// TIA Portal V16 program export: 11 tag tables, 23 data types, 17 data blocks, 38 code blocks (in call order from the OBs), 10 instance data blocks

VAR_GLOBAL   // PLC tag table "CONST"
END_VAR
VAR_GLOBAL CONSTANT   // user constants
   MAX_STEP_NUMB : Int := 50;
   MIN_STEP_NUMB : Int := 1;
   MAX_DEV_NUMB : Int := 16;
   MIN_DEV_NUMB : Int := 1;
   UF_CM_STANDBY : Int := 0;
   UF_CM_FILTRATION : Int := 2;
   UF_CM_START : Int := 1;
   UF_CM_HW : Int := 4;
   UF_CM_HW_A : Int := 5;
   UF_CM_CEB1 : Int := 6;
   UF_CM_CEB1_A : Int := 7;
   UF_CM_CEB2 : Int := 8;
   UF_CM_CEB2_A : Int := 9;
   UF_CM_STOP : Int := 3;
END_VAR

VAR_GLOBAL   // PLC tag table "Default tag table"
   System_Byte AT %MB1 : Byte;
   FirstScan AT %M1.0 : Bool;
   DiagStatusUpdate AT %M1.1 : Bool;
   AlwaysTRUE AT %M1.2 : Bool;
   AlwaysFALSE AT %M1.3 : Bool;
   Clock_Byte AT %MB0 : Byte;
   Clock_10Hz AT %M0.0 : Bool;
   Clock_5Hz AT %M0.1 : Bool;
   "Clock_2.5Hz" AT %M0.2 : Bool;
   Clock_2Hz AT %M0.3 : Bool;
   "Clock_1.25Hz" AT %M0.4 : Bool;
   Clock_1Hz AT %M0.5 : Bool;
   "Clock_0.625Hz" AT %M0.6 : Bool;
   "Clock_0.5Hz" AT %M0.7 : Bool;
   ClockOneSycle AT %MB2 : Byte;
   ClockOneCycle10HZ AT %M2.0 : Bool;
   ClockOneCycle5HZ AT %M2.1 : Bool;
   ClockOneCycle2_5HZ AT %M2.2 : Bool;
   ClockOneCycle2HZ AT %M2.3 : Bool;
   ClockOneCycle1_25HZ AT %M2.4 : Bool;
   ClockOneCycle1HZ AT %M2.5 : Bool;
   ClockOneCycle0_65HZ AT %M2.6 : Bool;
   ClockOneCycle0_5HZ AT %M2.7 : Bool;
END_VAR

VAR_GLOBAL   // PLC tag table "HW"
   PLC_RAW_DI AT %I0.0 : "PLC_HW_DI";
   PLC_RAW_DQ AT %Q0.0 : "PLC_HW_DQ";
   PLC_RAW_AI AT %I64.0 : "PLC_HW_AI";
   PLC_RAW_AQ AT %Q64.0 : "PLC_HW_AQ";
   ET_RAW_DI AT %I2.0 : "ET_HW_DI";
   ET_RAW_DQ AT %Q2.0 : "ET_HW_DQ";
   ET_RAW_AI AT %I68.0 : "ET_HW_AI";
   ET_RAW_AQ AT %Q68.0 : "ET_HW_AQ";
END_VAR
VAR_GLOBAL CONSTANT   // user constants
   PLC_DI : Int := 13;
   PLC_DQ : Int := 9;
   PLC_AI : Int := 1;
   PLC_AQ : Int := 1;
   ET_DI : Int := 79;
   ET_DQ : Int := 31;
   ET_AI : Int := 39;
   ET_AQ : Int := 7;
END_VAR

VAR_GLOBAL   // PLC tag table "A1_AI"
   aiDVA503_Pos AT %IW64 : Int;   // DVA503 Завдання
   aiDVA510_Pos AT %IW66 : Int;   // DVA510 Завдання
END_VAR
VAR_GLOBAL CONSTANT   // user constants
   "iwDVA-503_Setting" : Int := 0;
   "iwDVA-510_Setting" : Int := 1;
END_VAR

VAR_GLOBAL   // PLC tag table "A1_AQ"
   AO_DVA503_Setting AT %QW64 : Int;   // DVA503 Стан
   AO_DVA510_Setting AT %QW66 : Int;   // DVA510 Стан
END_VAR
VAR_GLOBAL CONSTANT   // user constants
   "qwDVA-503_Setting" : Int := 0;
   "qw_DVA-510_Setting" : Int := 1;
END_VAR

VAR_GLOBAL   // PLC tag table "A1_DI"
   iP301_Run AT %I0.0 : Bool;   // P301 Робота
   iP302_Run AT %I0.1 : Bool;   // P302 Робота
   iP1201_Run AT %I0.2 : Bool;   // P1201 Робота
   iP1202_Run AT %I0.3 : Bool;   // P1202 Робота
   iP1501_Run AT %I0.4 : Bool;   // P1501 Робота
   iP1502_Run AT %I0.5 : Bool;   // P1502 Робота
   iP70x_Ready AT %I0.6 : Bool;   // P70x Готовність
   iP701_Run AT %I0.7 : Bool;   // P701 Робота
   iP702_Run AT %I1.0 : Bool;   // P702 Робота
   iP201_Ready AT %I1.1 : Bool;   // P201 Готовність
   iP201_Run AT %I1.2 : Bool;   // P201 Робота
   iC501_Ready AT %I1.3 : Bool;   // C501 Готовність
   iStop AT %I1.4 : Bool;   // Аварійне вимикання
   iSF_Fail AT %I1.5 : Bool;   // Аварія захисних автоматів
END_VAR
VAR_GLOBAL CONSTANT   // user constants
   "iP-301_Run" : Int := 0;
   "iP-302_Run" : Int := 1;
   "iP-1201_Run" : Int := 2;
   "iP-1202_Run" : Int := 3;
   "iP-1501_Run" : Int := 4;
   "iP-1502_Run" : Int := 5;
   "iP-70x_Ready" : Int := 6;
   "iP-701_Run" : Int := 7;
   "iP-702_Run" : Int := 8;
   "iP-201_Ready" : Int := 9;
   "iP-201_Run" : Int := 10;
   "iC-501_Ready" : Int := 11;
   i_Stop : Int := 12;
   i_SF_Fail : Int := 13;
END_VAR

VAR_GLOBAL   // PLC tag table "A1_DQ"
   Tag_1 AT %Q0.0 : Bool;
   qP301_Start AT %Q0.1 : Bool;   // P301 Пуск
   qP302_Start AT %Q0.2 : Bool;   // P302 Пуск
   qP1201_Start AT %Q0.3 : Bool;   // P1201 Пуск
   qP1202_Start AT %Q0.4 : Bool;   // P1202 Пуск
   qP1501_Start AT %Q0.5 : Bool;   // P1501 Пуск
   qP1502_Start AT %Q0.6 : Bool;   // P1502 Пуск
   qP701_Start AT %Q0.7 : Bool;   // P701 Пуск
   qP702_Start AT %Q1.0 : Bool;   // P702 Пуск
   qP2001_Start AT %Q1.1 : Bool;   // P2001 Пуск
END_VAR
VAR_GLOBAL CONSTANT   // user constants
   iTag_1 : Int := 0;
   "qP-301_Start" : Int := 1;
   "qP-302_Start" : Int := 2;
   "qP-1201_Start" : Int := 3;
   "qP-1202_Start" : Int := 4;
   "qP-1501_Start" : Int := 5;
   "qP-1502_Start" : Int := 6;
   "qP-701_Start" : Int := 7;
   "qP-702_Start" : Int := 8;
   "qP-2001_Start" : Int := 9;
END_VAR

VAR_GLOBAL   // PLC tag table "A10_AI"
   aiLT201 AT %IW68 : Int;   // Рівень ємності TW201 LT201
   aiLT202 AT %IW70 : Int;   // Рівень ємності TW202 LT202
   aiPT301 AT %IW72 : Int;   // Тиск PS3 PT301
   aiPT401 AT %IW74 : Int;   // Тиск MDF4 PT401
   aiPT501 AT %IW76 : Int;   // Тиск повітря UF PT501
   aiPT502 AT %IW78 : Int;   // Тиск вхідної води UF PT502
   aiPT503 AT %IW80 : Int;   // Тиск фільтрата UF PT503
   aiPT504 AT %IW82 : Int;   // Тиск стічних вод UF PT504
   aiPT505 AT %IW84 : Int;   // Тиск вхідної води UF PT505
   aiPT506 AT %IW86 : Int;   // Тиск фільтрата UF PT506
   aiPT507 AT %IW88 : Int;   // Тиск стічних вод UF PT507
   aiLT601 AT %IW90 : Int;   // Рівень ємності TW601 LT601
   aiPT701 AT %IW92 : Int;   // Тиск PS7 PT701
   aiPT901 AT %IW94 : Int;   // Тиск насоса RO PT901
   aiPT902 AT %IW96 : Int;   // Тиск концентрата RO PT902
   aiLT1101 AT %IW98 : Int;   // Рівень ємності TW1101 LT1101
   aiPT1201 AT %IW100 : Int;   // Тиск PS12 PT1201
   aiPT1301 AT %IW102 : Int;   // Тиск насоса NF PT1301
   aiPT1302 AT %IW104 : Int;   // Тиск концентрата NF PT1302
   aiLT1401 AT %IW106 : Int;   // Рівень ємності TW1401 LT1401
   aiLT1402 AT %IW108 : Int;   // Рівень ємності TW1402 LT1402
   aiPT1501 AT %IW110 : Int;   // Тиск PS15 PT1501
   aiPT1701 AT %IW112 : Int;   // Тиск MCF17 PT1701
   aiLT1801 AT %IW114 : Int;   // Рівень ємності TW1801 LT1801
   aiFM501 AT %IW116 : Int;   // Витрата вхідної води UF FM501
   aiFM502 AT %IW118 : Int;   // Витрата вхідної води UF FM502
   aiFM901 AT %IW120 : Int;   // Витрата пермеату RO FM901
   aiFM902 AT %IW122 : Int;   // Витрата концентрату RO FM902
   aiFM1301 AT %IW124 : Int;   // Витрата пермеату NF FM901
   aiFM1302 AT %IW126 : Int;   // Витрата концентрату NF FM902
   aiORP801 AT %IW128 : Int;   // ORP води на UF ORP801
   aiCDI901 AT %IW130 : Int;   // Електропровідність пермеату RO CDI901
   aiCDI1301 AT %IW132 : Int;   // Електропровідність пермеату RO CD1301
   aiCDI1302 AT %IW134 : Int;   // Електропровідність після змішування CD1302
   aiCDI1801 AT %IW136 : Int;   // Електропровідність стічних вод CD1801
   PIW74_Reserve AT %IW138 : Int;   // Резерв
   PIW76_Reserve AT %IW140 : Int;   // Резерв
   PIW78_Reserve AT %IW142 : Int;   // Резерв
   PIW80_Reserve AT %IW144 : Int;   // Резерв
   PIW82_Reserve AT %IW146 : Int;   // Резерв
END_VAR
VAR_GLOBAL CONSTANT   // user constants
   iwLT201 : Int := 0;
   iwLT202 : Int := 1;
   iwPT301 : Int := 2;
   iwPT401 : Int := 3;
   iwPT501 : Int := 4;
   iwPT502 : Int := 5;
   iwPT503 : Int := 6;
   iwPT504 : Int := 7;
   iwPT505 : Int := 8;
   iwPT506 : Int := 9;
   iwPT507 : Int := 10;
   iwLT601 : Int := 11;
   iwPT701 : Int := 12;
   iwPT901 : Int := 13;
   iwPT902 : Int := 14;
   iwLT1101 : Int := 15;
   iwPT1201 : Int := 16;
   iwPT1301 : Int := 17;
   iwPT1302 : Int := 18;
   iwLT1401 : Int := 19;
   iwLT1402 : Int := 20;
   iwPT1501 : Int := 21;
   iwPT1701 : Int := 22;
   iwLT1801 : Int := 23;
   iwFM501 : Int := 24;
   iwFM502 : Int := 25;
   iwFM901 : Int := 26;
   iwFM902 : Int := 27;
   iwFM1301 : Int := 28;
   iwFM1302 : Int := 29;
   iwORP801 : Int := 30;
   iwCDI901 : Int := 31;
   iwCDI1301 : Int := 32;
   iwCDI1302 : Int := 33;
   iwCDI1801 : Int := 34;
   iw74_Reserve : Int := 35;
   iw76_Reserve : Int := 36;
   iw78_Reserve : Int := 37;
   iw80_Reserve : Int := 38;
   iw82_Reserve : Int := 39;
END_VAR

VAR_GLOBAL   // PLC tag table "A10_AQ"
   aqDP101 AT %QW68 : Int;   // DP101 Завдання
   aqDP502 AT %QW70 : Int;   // DP502 Завдання
   aqDP501 AT %QW72 : Int;   // DP501 Завдання
   aqDP801 AT %QW74 : Int;   // DP801 Завдання
   aqDP802 AT %QW76 : Int;   // DP802 Завдання
   aqDP803 AT %QW78 : Int;   // DP803 Завдання
   aqDP1001 AT %QW80 : Int;   // DP1001 Завдання
   PQW18_Reserve AT %QW82 : Int;   // Резерв
END_VAR
VAR_GLOBAL CONSTANT   // user constants
   "qwDP-101" : Int := 0;
   "qwDP-502" : Int := 1;
   "qwDP-501" : Int := 2;
   "qwDP-801" : Int := 3;
   "qwDP-802" : Int := 4;
   "qwDP-803" : Int := 5;
   "qwDP-1001" : Int := 6;
   qw18_Reserve : Int := 7;
END_VAR

VAR_GLOBAL   // PLC tag table "A10_DI"
   iDP101_Run AT %I2.0 : Bool;   // DP101 Робота
   iDP101_Fail AT %I2.1 : Bool;   // DP101 Аварія
   iDP502_Run AT %I2.2 : Bool;   // DP502 Робота
   iDP502_Fail AT %I2.3 : Bool;   // DP502 Аварія
   iDP501_Run AT %I2.4 : Bool;   // DP501 Робота
   iDP501_Fail AT %I2.5 : Bool;   // DP501 Аварія
   iDP801_Run AT %I2.6 : Bool;   // DP801 Робота
   iDP801_Fail AT %I2.7 : Bool;   // DP801 Аварія
   iDP802_Run AT %I3.0 : Bool;   // DP802 Робота
   iDP802_Fail AT %I3.1 : Bool;   // DP802 Аварія
   iDP803_Run AT %I3.2 : Bool;   // DP803 Робота
   iDP803_Fail AT %I3.3 : Bool;   // DP803 Аварія
   iDP1001_Run AT %I3.4 : Bool;   // DP1001 Робота
   iDP1001_Fail AT %I3.5 : Bool;   // DP1001 Аварія
   iUV1601_Fail AT %I3.6 : Bool;   // UV1601 Аварія
   "I3.7_Reserve" AT %I3.7 : Bool;   // Резерв
   iPS901 AT %I4.0 : Bool;   // Тиск на вході насоса зворотнього осмоса PS901
   iPS902 AT %I4.1 : Bool;   // Тиск перемеата зворотнього осмоса PS902
   iPS1301 AT %I4.2 : Bool;   // Тиск на вході насоса нанофільтрації PS1301
   iPS1302 AT %I4.3 : Bool;   // Тиск перемеата нанофільтрації PS1302
   iFL501 AT %I4.4 : Bool;   // Витрата повітря на промивку ультрафільтрації FL501
   iFL901 AT %I4.5 : Bool;   // Витрата рециклу зворотнього осмоса FL901
   iFL1301 AT %I4.6 : Bool;   // Витрата рециклу нанофільтрації FL1301
   iFM201 AT %I4.7 : Bool;   // Витрата вхідної води FM201
   iFM1201 AT %I5.0 : Bool;   // Витрата пермеату на споживоча FM1201
   iFM1701 AT %I5.1 : Bool;   // Витрата нанофільтрату на споживоча FM1701
   iFM1801 AT %I5.2 : Bool;   // Витрата стічних вод FM1801
   iFM501 AT %I5.3 : Bool;   // Витрата вхідної води UF FM501
   iFM502 AT %I5.4 : Bool;   // Витрата вхідної води UF FM502
   iFM901 AT %I5.5 : Bool;   // Витрата пермеату RO FM901
   iFM902 AT %I5.6 : Bool;   // Витрата концентрату RO FM902
   iFM1301 AT %I5.7 : Bool;   // Витрата пермеату NF FM1301
   iFM1302 AT %I6.0 : Bool;   // Витрата концентрату NF FM1302
   iDVA501_closed AT %I6.1 : Bool;   // Клапан DVA501 закрит
   iDVA501_open AT %I6.2 : Bool;   // Клапан DVA501 открит
   iDVA502_closed AT %I6.3 : Bool;   // Клапан DVA502 закрит
   iDVA502_open AT %I6.4 : Bool;   // Клапан DVA502 открит
   iDVA504_closed AT %I6.5 : Bool;   // Клапан DVA504 закрит
   iDVA504_open AT %I6.6 : Bool;   // Клапан DVA504 открит
   "I6.7_reserve" AT %I6.7 : Bool;   // Резерв
   iDVA505_closed AT %I7.0 : Bool;   // Клапан DVA505 закрит
   iDVA505_open AT %I7.1 : Bool;   // Клапан DVA505 открит
   iDVA506_closed AT %I7.2 : Bool;   // Клапан DVA506 закрит
   iDVA506_open AT %I7.3 : Bool;   // Клапан DVA506 открит
   iDVA507_closed AT %I7.4 : Bool;   // Клапан DVA507 закрит
   iDVA507_open AT %I7.5 : Bool;   // Клапан DVA507 открит
   iDVA508_closed AT %I7.6 : Bool;   // Клапан DVA508 закрит
   iDVA508_open AT %I7.7 : Bool;   // Клапан DVA508 открит
   iDVA509_closed AT %I8.0 : Bool;   // Клапан DVA509 закрит
   iDVA509_open AT %I8.1 : Bool;   // Клапан DVA509 открит
   iDVA511_closed AT %I8.2 : Bool;   // Клапан DVA511 закрит
   iDVA511_open AT %I8.3 : Bool;   // Клапан DVA511 открит
   iDVA512_closed AT %I8.4 : Bool;   // Клапан DVA512 закрит
   iDVA512_open AT %I8.5 : Bool;   // Клапан DVA512 открит
   iDVA513_closed AT %I8.6 : Bool;   // Клапан DVA513 закрит
   iDVA513_open AT %I8.7 : Bool;   // Клапан DVA513 открит
   iDVA514_closed AT %I9.0 : Bool;   // Клапан DVA514 закрит
   iDVA514_open AT %I9.1 : Bool;   // Клапан DVA514 открит
   iDVA515_closed AT %I9.2 : Bool;   // Клапан DVA515 закрит
   iDVA515_open AT %I9.3 : Bool;   // Клапан DVA515 открит
   iDVA516_closed AT %I9.4 : Bool;   // Клапан DVA516 закрит
   iDVA516_open AT %I9.5 : Bool;   // Клапан DVA516 открит
   iDVA1801_closed AT %I9.6 : Bool;   // Клапан DVA1801 закрит
   iDVA1801_open AT %I9.7 : Bool;   // Клапан DVA1801 открит
   iP3xx_Stop AT %I10.0 : Bool;   // P3xx Аварійне вимиканя
   iP901_Stop AT %I10.1 : Bool;   // P901 Аварійне вимиканя
   iP1301_Stop AT %I10.2 : Bool;   // P13xx Аварійне вимиканя
   iP12xx_Stop AT %I10.3 : Bool;   // P12xx Аварійне вимиканя
   iP15xx_Stop AT %I10.4 : Bool;   // P15xx Аварійне вимиканя
   iP7xx_Stop AT %I10.5 : Bool;   // P7xx Аварійне вимиканя
   iP2001_Stop AT %I10.6 : Bool;   // P2001 Аварійне вимиканя
   "I10.7_reserve" AT %I10.7 : Bool;   // Резерв
   "I11.0_reserve" AT %I11.0 : Bool;   // Резерв
   "I11.1_reserve" AT %I11.1 : Bool;   // Резерв
   "I11.2_reserve" AT %I11.2 : Bool;   // Резерв
   "I11.3_reserve" AT %I11.3 : Bool;   // Резерв
   "I11.4_reserve" AT %I11.4 : Bool;   // Резерв
   "I11.5_reserve" AT %I11.5 : Bool;   // Резерв
   "I11.6_reserve" AT %I11.6 : Bool;   // Резерв
   "I11.7_reserve" AT %I11.7 : Bool;   // Резерв
END_VAR
VAR_GLOBAL CONSTANT   // user constants
   "iDP-101_Run" : Int := 0;
   "iDP-101_Fail" : Int := 1;
   "iDP-502_Run" : Int := 2;
   "iDP-502_Fail" : Int := 3;
   "iDP-501_Run" : Int := 4;
   "iDP-501_Fail" : Int := 5;
   "iDP-801_Run" : Int := 6;
   "iDP-801_Fail" : Int := 7;
   "iDP-802_Run" : Int := 8;
   "iDP-802_Fail" : Int := 9;
   "iDP-803_Run" : Int := 10;
   "iDP-803_Fail" : Int := 11;
   "iDP-1001_Run" : Int := 12;
   "iDP-1001_Fail" : Int := 13;
   "iUV-1601_Fail" : Int := 14;
   "I3.7_res" : Int := 15;
   i_PS901 : Int := 16;
   i_PS902 : Int := 17;
   i_PS1301 : Int := 18;
   i_PS1302 : Int := 19;
   i_FL501 : Int := 20;
   i_FL901 : Int := 21;
   i_FL1301 : Int := 22;
   i_FM201 : Int := 23;
   i_FM1201 : Int := 24;
   i_FM1701 : Int := 25;
   i_FM1801 : Int := 26;
   i_FM501 : Int := 27;
   i_FM502 : Int := 28;
   i_FM901 : Int := 29;
   i_FM902 : Int := 30;
   i_FM1301 : Int := 31;
   i_FM1302 : Int := 32;
   "iDVA-501_closed" : Int := 33;
   "iDVA-501_open" : Int := 34;
   "iDVA-502_closed" : Int := 35;
   "iDVA-502_open" : Int := 36;
   "iDVA-504_closed" : Int := 37;
   "iDVA-504_open" : Int := 38;
   "I6.7_res" : Int := 39;
   "iDVA-505_closed" : Int := 40;
   "iDVA-505_open" : Int := 41;
   "iDVA-506_closed" : Int := 42;
   "iDVA-506_open" : Int := 43;
   "iDVA-507_closed" : Int := 44;
   "iDVA-507_open" : Int := 45;
   "iDVA-508_closed" : Int := 46;
   "iDVA-508_open" : Int := 47;
   "iDVA-509_closed" : Int := 48;
   "iDVA-509_open" : Int := 49;
   "iDVA-511_closed" : Int := 50;
   "iDVA-511_open" : Int := 51;
   "iDVA-512_closed" : Int := 52;
   "iDVA-512_open" : Int := 53;
   "iDVA-513_closed" : Int := 54;
   "iDVA-513_open" : Int := 55;
   "iDVA-514_closed" : Int := 56;
   "iDVA-514_open" : Int := 57;
   "iDVA-515_closed" : Int := 58;
   "iDVA-515_open" : Int := 59;
   "iDVA-516_closed" : Int := 60;
   "iDVA-516_open" : Int := 61;
   "iDVA-1801_closed" : Int := 62;
   "iDVA-1801_open" : Int := 63;
   "iP-3xx_Stop" : Int := 64;
   "iP-901_Stop" : Int := 65;
   "iP-1301_Stop" : Int := 66;
   "iP-12xx_Stop" : Int := 67;
   "iP-15xx_Stop" : Int := 68;
   "iP-7xx_Stop" : Int := 69;
   "iP-2001_Stop" : Int := 70;
   "I10.7_res" : Int := 71;
   "I11.0_res" : Int := 72;
   "I11.1_res" : Int := 73;
   "I11.2_res" : Int := 74;
   "I11.3_res" : Int := 75;
   "I11.4_res" : Int := 76;
   "I11.5_res" : Int := 77;
   "I11.6_res" : Int := 78;
   "I11.7_res" : Int := 79;
END_VAR

VAR_GLOBAL   // PLC tag table "A10_DQ"
   qDP101_Start AT %Q2.0 : Bool;   // DP101 Пуск
   qDP502_Start AT %Q2.1 : Bool;   // DP502 Пуск
   qDP501_Start AT %Q2.2 : Bool;   // DP501 Пуск
   qDP801_Start AT %Q2.3 : Bool;   // DP801 Пуск
   qDP802_Start AT %Q2.4 : Bool;   // DP802 Пуск
   qDP803_Start AT %Q2.5 : Bool;   // DP803 Пуск
   qDP1001_Start AT %Q2.6 : Bool;   // DP1001 Пуск
   "Q2.7_Reserve" AT %Q2.7 : Bool;   // Резерв
   qDVM201_Open AT %Q3.0 : Bool;   // DVM201 Відкрити
   qSOV801_Open AT %Q3.1 : Bool;   // SOV801 Відкрити
   qSOV901_Open AT %Q3.2 : Bool;   // SOV901 Відкрити
   qSOV902_Open AT %Q3.3 : Bool;   // SOV902 Відкрити
   qSOV1301_Open AT %Q3.4 : Bool;   // SOV1301 Відкрити
   qSOV1302_Open AT %Q3.5 : Bool;   // SOV1302 Відкрити
   qSOV1303_Open AT %Q3.6 : Bool;   // SOV1303 Відкрити
   "Q3.7_Reserve" AT %Q3.7 : Bool;   // Резерв
   qDVA501_Open AT %Q4.0 : Bool;   // DVA501 Відкрити
   qDVA502_Open AT %Q4.1 : Bool;   // DVA502 Відкрити
   qDVA504_Open AT %Q4.2 : Bool;   // DVA504 Відкрити
   qDVA505_Open AT %Q4.3 : Bool;   // DVA505 Відкрити
   qDVA506_Open AT %Q4.4 : Bool;   // DVA506 Відкрити
   qDVA507_Open AT %Q4.5 : Bool;   // DVA507 Відкрити
   qDVA508_Open AT %Q4.6 : Bool;   // DVA508 Відкрити
   qDVA509_Open AT %Q4.7 : Bool;   // DVA509 Відкрити
   qDVA511_Open AT %Q5.0 : Bool;   // DVA511 Відкрити
   qDVA512_Open AT %Q5.1 : Bool;   // DVA512 Відкрити
   qDVA513_Open AT %Q5.2 : Bool;   // DVA513 Відкрити
   qDVA514_Open AT %Q5.3 : Bool;   // DVA514 Відкрити
   qDVA515_Open AT %Q5.4 : Bool;   // DVA515 Відкрити
   qDVA516_Open AT %Q5.5 : Bool;   // DVA516 Відкрити
   qDVA1801_Open AT %Q5.6 : Bool;   // DVA1801 Відкрити
   qMDF4 AT %Q5.7 : Bool;   // Фільтр дисковий
END_VAR
VAR_GLOBAL CONSTANT   // user constants
   "qDP-101_Start" : Int := 0;
   "qDP-502_Start" : Int := 1;
   "qDP-501_Start" : Int := 2;
   "qDP-801_Start" : Int := 3;
   "qDP-802_Start" : Int := 4;
   "qDP-803_Start" : Int := 5;
   "qDP-1001_Start" : Int := 6;
   "Q2.7_res" : Int := 7;
   "qDVM-201_Open" : Int := 8;
   "qSOV-801_Open" : Int := 9;
   "qSOV-901_Open" : Int := 10;
   "qSOV-902_Open" : Int := 11;
   "qSOV-1301_Open" : Int := 12;
   "qSOV-1302_Open" : Int := 13;
   "qSOV-1303_Open" : Int := 14;
   "Q3.7_res" : Int := 15;
   "qDVA-501_Open" : Int := 16;
   "qDVA-502_Open" : Int := 17;
   "qDVA-504_Open" : Int := 18;
   "qDVA-505_Open" : Int := 19;
   "qDVA-506_Open" : Int := 20;
   "qDVA-507_Open" : Int := 21;
   "qDVA-508_Open" : Int := 22;
   "qDVA-509_Open" : Int := 23;
   "qDVA-511_Open" : Int := 24;
   "qDVA-512_Open" : Int := 25;
   "qDVA-513_Open" : Int := 26;
   "qDVA-514_Open" : Int := 27;
   "qDVA-515_Open" : Int := 28;
   "qDVA-516_Open" : Int := 29;
   "qDVA-1801_Open" : Int := 30;
   "Q5.7_res" : Int := 31;
END_VAR

TYPE "Ai"
// stored: IsFailsafeCompliant false
   STRUCT
      emMax_En { ExternalAccessible := 'False'; ExternalVisible := 'False'; ExternalWritable := 'False'; S7_SetPoint := 'True'} : Bool;   // Аварийный верхний 1-проверять
      emMin_En { ExternalAccessible := 'False'; ExternalVisible := 'False'; ExternalWritable := 'False'; S7_SetPoint := 'True'} : Bool;   // Аварийный нижний 1-проверять
      wrnMax_En { ExternalAccessible := 'False'; ExternalVisible := 'False'; ExternalWritable := 'False'; S7_SetPoint := 'True'} : Bool;   // Предупредительный верхний 1-проверять
      wrnMin_En { ExternalAccessible := 'False'; ExternalVisible := 'False'; ExternalWritable := 'False'; S7_SetPoint := 'True'} : Bool;   // Предупредительный нижний 1-проверять
      curEmMax { ExternalAccessible := 'False'; ExternalVisible := 'False'; ExternalWritable := 'False'} : Bool;   // В данный момент значение выше аварийного максимума
      curEmMin { ExternalAccessible := 'False'; ExternalVisible := 'False'; ExternalWritable := 'False'} : Bool;   // В данный момент значение ниже аварийного минимума
      curWnMax { ExternalAccessible := 'False'; ExternalVisible := 'False'; ExternalWritable := 'False'} : Bool;   // В данный момент значение выше предупредительного максимума
      curWnMin { ExternalAccessible := 'False'; ExternalVisible := 'False'; ExternalWritable := 'False'} : Bool;   // В данный момент значение ниже предупредительного минимума
      emMax { ExternalAccessible := 'False'; ExternalVisible := 'False'; ExternalWritable := 'False'} : Bool;   // Сработала сигнализация - аварийный максимум
      emMin { ExternalAccessible := 'False'; ExternalVisible := 'False'; ExternalWritable := 'False'} : Bool;   // Сработала сигнализация - аварийный минимум
      wnMax { ExternalAccessible := 'False'; ExternalVisible := 'False'; ExternalWritable := 'False'} : Bool;   // Сработала сигнализация - предупредительный максимум
      wnMin { ExternalAccessible := 'False'; ExternalVisible := 'False'; ExternalWritable := 'False'} : Bool;   // Сработала сигнализация - предупредительный минимум
      Err : Bool;   // Наличие ошибок канала / Налицие ошибок канала
      badParam { ExternalVisible := 'False'} : Bool;   // Неправильные параметры
      overFlow { ExternalVisible := 'False'} : Bool;   // Перегрузка канала
      wireBreak { ExternalVisible := 'False'} : Bool;   // Обрыв провода
      SimEnable { S7_SetPoint := 'True'} : Bool;   // Включение симуляции
      disableParLessZero { S7_SetPoint := 'True'} : Bool := 1;   // 1-Запрет значений меньше нуля, типа плавающих значений
      modeAck { S7_SetPoint := 'True'} : Bool := 1;   // 1-сброс по общему сбросу аварий, 0-сброс после исчезновения условия
      ackAll : Bool;   // сброс всех событий
      ack { ExternalVisible := 'False'} : Byte;   // Байт сброса ошибок
      State : Word;   // Код качества
      Par_code { ExternalVisible := 'False'} : Int;   // Код канала
      Par : Real;   // Значение параметра в технологических единицах
      rngUpLm { ExternalVisible := 'False'; S7_SetPoint := 'True'} : Real := 200.0;   // Максимум диапазона измерения
      rngLwLm { ExternalVisible := 'False'; S7_SetPoint := 'True'} : Real;   // Минимум диапазона измерения
      emrMax { ExternalVisible := 'False'; S7_SetPoint := 'True'} : Real := 190.0;   // Технологический верхний аварийный предел
      emrMaxTime { ExternalVisible := 'False'; S7_SetPoint := 'True'} : Real := 5.0;   // Время задержки для срабатывания аварии по Аварийному верхнему пределу
      emrMin { ExternalVisible := 'False'; S7_SetPoint := 'True'} : Real := 10.0;   // Технологический нижний аварийный предел
      emrMinTime { ExternalVisible := 'False'; S7_SetPoint := 'True'} : Real := 5.0;   // Время задержки для срабатывания аварии по Аварийному нижниму пределу
      wrnMax { ExternalVisible := 'False'; S7_SetPoint := 'True'} : Real := 150.0;   // Технологический верхний предупредительный предел
      wrnMaxTime { ExternalVisible := 'False'; S7_SetPoint := 'True'} : Real := 5.0;   // Время задержки для срабатывания аварии по Предупредительному верхнему пределу
      wrnMin { ExternalVisible := 'False'; S7_SetPoint := 'True'} : Real := 20.0;   // Технологический нижний предупредительный предел
      wrnMinTime { ExternalVisible := 'False'; S7_SetPoint := 'True'} : Real := 5.0;   // Время задержки для срабатывания аварии по Предупредительному нижниму пределу
      Par_mA { ExternalVisible := 'False'} : Real;   // Значение параметра в мА
      SimValue { ExternalVisible := 'False'} : Real;   // Значение симуляции
      curTimeEmrMin { ExternalAccessible := 'False'; ExternalVisible := 'False'; ExternalWritable := 'False'} : Real;   // Текуще значение таймера
      curTimeWrnMin { ExternalAccessible := 'False'; ExternalVisible := 'False'; ExternalWritable := 'False'} : Real;   // Текуще значение таймера
      curTimeWrnMax { ExternalAccessible := 'False'; ExternalVisible := 'False'; ExternalWritable := 'False'} : Real;   // Текуще значение таймера
      curTimeEmrMax { ExternalAccessible := 'False'; ExternalVisible := 'False'; ExternalWritable := 'False'} : Real;   // Текуще значение таймера
      Spare_0 { ExternalAccessible := 'False'; ExternalVisible := 'False'; ExternalWritable := 'False'} : Word;
      Spare_1 { ExternalAccessible := 'False'; ExternalVisible := 'False'; ExternalWritable := 'False'} : Word;
      Spare_2 { ExternalAccessible := 'False'; ExternalVisible := 'False'; ExternalWritable := 'False'} : Word;
      Spare_3 { ExternalAccessible := 'False'; ExternalVisible := 'False'; ExternalWritable := 'False'} : Word;
      Spare_4 { ExternalAccessible := 'False'; ExternalVisible := 'False'; ExternalWritable := 'False'} : Word;
      Spare_5 { ExternalAccessible := 'False'; ExternalVisible := 'False'; ExternalWritable := 'False'} : Word;
      Spare_6 { ExternalAccessible := 'False'; ExternalVisible := 'False'; ExternalWritable := 'False'} : Word;
      Spare_7 { ExternalAccessible := 'False'; ExternalVisible := 'False'; ExternalWritable := 'False'} : Word;
      Spare_8 { ExternalAccessible := 'False'; ExternalVisible := 'False'; ExternalWritable := 'False'} : Word;
      Spare_9 { ExternalAccessible := 'False'; ExternalVisible := 'False'; ExternalWritable := 'False'} : Word;
      Spare_10 { ExternalAccessible := 'False'; ExternalVisible := 'False'; ExternalWritable := 'False'} : Word;
      Spare_11 { ExternalAccessible := 'False'; ExternalVisible := 'False'; ExternalWritable := 'False'} : Word;
   END_STRUCT;
END_TYPE

TYPE "Av"
// stored: IsFailsafeCompliant false
   STRUCT
      mode : Bool;   // 0-ручной, 1-авто
      cmAuto { ExternalAccessible := 'False'; ExternalVisible := 'False'; ExternalWritable := 'False'} : Bool;   // авто команда
      cmHand : Bool;   // ручная команда
      block { ExternalAccessible := 'False'; ExternalVisible := 'False'; ExternalWritable := 'False'} : Bool;   // Внешняя блокировка
      error { ExternalAccessible := 'False'; ExternalVisible := 'False'; ExternalWritable := 'False'} : Bool;   // Общая ошибка
      checkOC { S7_SetPoint := 'True'} : Bool;   // Проверка концевиков
      outCmStart { ExternalAccessible := 'False'; ExternalVisible := 'False'; ExternalWritable := 'False'} : Bool;   // Программный выход
      st : Word;   // Состояние
      tOpen { S7_SetPoint := 'True'} : Int := 10;   // Время открытия, сек
      tClose { S7_SetPoint := 'True'} : Int := 10;   // Время закрытия, сек
      ack { ExternalAccessible := 'False'; ExternalVisible := 'False'; ExternalWritable := 'False'} : Word;
      spare_0 { ExternalAccessible := 'False'; ExternalVisible := 'False'; ExternalWritable := 'False'} : Word;
      spare_1 { ExternalAccessible := 'False'; ExternalVisible := 'False'; ExternalWritable := 'False'} : DInt;
   END_STRUCT;
END_TYPE

TYPE "DPump"
// stored: IsFailsafeCompliant false
   STRUCT
      mode : Bool;   // 1-ручной, 0-авто
      cmAuto { ExternalAccessible := 'False'; ExternalVisible := 'False'; ExternalWritable := 'False'} : Bool;   // авто команда
      cmHand : Bool;   // ручная команда
      block { ExternalAccessible := 'False'; ExternalVisible := 'False'; ExternalWritable := 'False'} : Bool;   // Внешняя блокировка
      service : Bool;   // Сервисный режим
      error { ExternalAccessible := 'False'; ExternalVisible := 'False'; ExternalWritable := 'False'} : Bool;   // Наличие любой ошибки
      showButton : Bool;   // 0- Показать, 1 - Скрыть
      feedBack { S7_SetPoint := 'True'} : Bool;   // Обратная связь
      st : Word;   // Состояние
      startTime { S7_SetPoint := 'True'} : Int := 5;   // Время запуска, сек
      stopTime { S7_SetPoint := 'True'} : Int := 5;   // Время останова, сек
      outCmStart { ExternalAccessible := 'False'; ExternalVisible := 'False'; ExternalWritable := 'False'} : Bool;   // Программный выход запуска насоса
      ack { ExternalAccessible := 'False'; ExternalVisible := 'False'; ExternalWritable := 'False'} : Word;   // Резерв
      spare1 : Word;
   END_STRUCT;
END_TYPE

TYPE "FREQ_COUNTER"
// stored: IsFailsafeCompliant false
   STRUCT
      litrsPerPuls : UInt;
      prewHour : UInt;
      curHour : UInt;
      prewDay : UDInt;
      curDay : UDInt;
      all : UDInt;
      rst : Bool;
   END_STRUCT;
END_TYPE

TYPE "PropDosing"
// stored: IsFailsafeCompliant false
   STRUCT
      FE : Real;   // расход для определения дозы
      max : Real;   // доза при 20 мА
      spAuto { S7_SetPoint := 'True'} : Real := 5.0;   // задание авто (г/м3)
      spHand { S7_SetPoint := 'True'} : Real;   // задание ручное (л/ч)
      outSP : Real;   // Производительность (%)
      outPQW : Int;   // Выход на PQW
      outLPH : Real;   // Выход (л/ч)
      mode : Bool;   // 0-ручной,1-авто
      enableFix { ExternalVisible := 'False'; ExternalWritable := 'False'} : Bool;   // включение фиксированного задания
      density { S7_SetPoint := 'True'} : Real;
      outmA : Real;
      minFE { S7_SetPoint := 'True'} : Real;
      fixSP { ExternalVisible := 'False'; ExternalWritable := 'False'} : Real;   // задание от пид регулятора
      spareDint : DInt;
   END_STRUCT;
END_TYPE

TYPE "Pump"
// stored: IsFailsafeCompliant false
   STRUCT
      mode : Bool;   // 1-ручной, 0-авто
      cmAuto { ExternalAccessible := 'False'; ExternalVisible := 'False'; ExternalWritable := 'False'} : Bool;   // авто команда
      cmHand : Bool;   // ручная команда
      block { ExternalAccessible := 'False'; ExternalVisible := 'False'; ExternalWritable := 'False'} : Bool;   // Внешняя блокировка
      service : Bool;   // Сервисный режим
      error { ExternalAccessible := 'False'; ExternalVisible := 'False'; ExternalWritable := 'False'} : Bool;   // Наличие любой ошибки
      showButton : Bool;   // 0- Показать, 1 - Скрыть
      feedBack { S7_SetPoint := 'True'} : Bool;   // Обратная связь
      st : Word;   // Состояние
      startTime { S7_SetPoint := 'True'} : Int := 5;   // Время запуска, сек
      stopTime { S7_SetPoint := 'True'} : Int := 5;   // Время останова, сек
      outCmStart { ExternalAccessible := 'False'; ExternalVisible := 'False'; ExternalWritable := 'False'} : Bool;   // Программный выход запуска насоса
      resetTimeWork : Bool;
      ack { ExternalAccessible := 'False'; ExternalVisible := 'False'; ExternalWritable := 'False'} : Word;
      blockDetail : Word;   // Подробности блокировки
      timeWork : UDInt;
      tWorkString : String;
   END_STRUCT;
END_TYPE

TYPE "SeqStep"
// stored: IsFailsafeCompliant false
   STRUCT
      StepDev { S7_SetPoint := 'True'} : Array[1..32] of Word;
      StepDelay { S7_SetPoint := 'True'} : Array[1..32] of Time;
      initDev : Word;
      AlgN : Int;
      nStartStep { S7_SetPoint := 'True'} : Int := 1;
   END_STRUCT;
END_TYPE

TYPE "UF_COMMANDS"
// stored: IsFailsafeCompliant false
   STRUCT
      Start : Bool;
      Stop : Bool;
      HW : Bool;
      HW_A : Bool;
      CEB1 : Bool;
      CEB1_A : Bool;
      CEB2 : Bool;
      CEB2_A : Bool;
   END_STRUCT;
END_TYPE

TYPE "UF_COUNTERS"
// stored: IsFailsafeCompliant false
   STRUCT
      HDPW : UInt;   // High delta preassure wash
      HW : UInt;
      CEB1 : UInt;
      CEB2 : UInt;
   END_STRUCT;
END_TYPE

TYPE "UF_FLAGS"
// stored: IsFailsafeCompliant false
   STRUCT
      StandBy : Bool;
      Stop : Bool;
      Filtration : Bool;
      Start : Bool;
      HW : Bool;
      HW_A : Bool;
      CEB1 : Bool;
      CEB1_A : Bool;
      CEB2 : Bool;
      CEB2_A : Bool;
      Err : Bool;
      ErrWork : Bool;
      ErrHW : Bool;
      ErrCEB1 : Bool;
      ErrCEB2 : Bool;
      ErrHDP : Bool;
   END_STRUCT;
END_TYPE

TYPE "UF_PARAMETRS"
// stored: IsFailsafeCompliant false
   STRUCT
      Sf : Real;   // Filtration square m2
      flux : Real;
      dP : Real;   // Delta preassure
      Rec : Real;   // Recovery
      Ts : UInt;   // Step time
      Tf : UDInt;   // Filtration time
   END_STRUCT;
END_TYPE

TYPE "UZ_Data"
// stored: IsFailsafeCompliant false
   STRUCT
      Ready { ExternalAccessible := 'False'; ExternalVisible := 'False'; ExternalWritable := 'False'} : Bool;   // Drive ready to start
      Fault { ExternalAccessible := 'False'; ExternalVisible := 'False'; ExternalWritable := 'False'} : Bool;   // Fault is present. Trip or Trip lock
      Warning { ExternalAccessible := 'False'; ExternalVisible := 'False'; ExternalWritable := 'False'} : Bool;   // Warning present
      Running : Bool;   // Drive is started but not necessarily running on reference speed.
      Run_On_ref { ExternalAccessible := 'False'; ExternalVisible := 'False'; ExternalWritable := 'False'} : Bool;   // Running on reference
      MotorCurrent : Real;   // Actual motor Current
      MotorPower : Real;   // Motor Power
      MAV : Real;   // Main Actual Value read from Drive 0 - 100.00%
      comErr { ExternalAccessible := 'False'; ExternalVisible := 'False'; ExternalWritable := 'False'} : Int;   // Result of DPRD_DAT 0=No error
      ErrorConnection : Bool;   // Present Error DPRD_DAT
   END_STRUCT;
END_TYPE

TYPE "digitalSensor"
// stored: IsFailsafeCompliant false
   STRUCT
      simMode { ExternalAccessible := 'False'; ExternalVisible := 'False'; ExternalWritable := 'False'} : Bool;   // 0-auto, 1-hand
      direction { ExternalAccessible := 'False'; ExternalVisible := 'False'; ExternalWritable := 'False'} : Bool;   // 0-прямой, 1-инверсный
      simOn { ExternalAccessible := 'False'; ExternalVisible := 'False'; ExternalWritable := 'False'} : Bool;   // 1-On
      out : Bool;   // 0-nomr, 1-alarm
      statePRG { ExternalAccessible := 'False'; ExternalVisible := 'False'; ExternalWritable := 'False'} : Bool;   // программное состояние в зависимости от режим
      inHW { ExternalAccessible := 'False'; ExternalVisible := 'False'; ExternalWritable := 'False'} : Bool;
      enableDetection { ExternalAccessible := 'False'; ExternalVisible := 'False'; ExternalWritable := 'False'} : Bool;   // 1-включить детектирование аварии
      ackBit : Bool;   // индивидуальный бит сброса аварии
      delay { ExternalAccessible := 'False'; ExternalVisible := 'False'; ExternalWritable := 'False'} : Real := 5.0;   // задержка
      curTime { ExternalAccessible := 'False'; ExternalVisible := 'False'; ExternalWritable := 'False'} : Real;   // Current time
   END_STRUCT;
END_TYPE

TYPE "setPID"
// stored: IsFailsafeCompliant false
   STRUCT
      spAuto { S7_SetPoint := 'True'} : Real;
      spHand : Real;
      TI { S7_SetPoint := 'True'} : Real := 10.0;
      Gain { S7_SetPoint := 'True'} : Real := 2.0;
      min { S7_SetPoint := 'True'} : Real := 30.0;
      max { S7_SetPoint := 'True'} : Real := 100.0;
      dead { S7_SetPoint := 'True'} : Real := 0.1;
      outPID : Real;
      cmFixSP : Bool;
      cmFreeze : Bool;
      cmStartSP : Bool;
      spareByte : Byte;
      fixSP { S7_SetPoint := 'True'} : Real;
      spStart : Real;
      spare_2 : DInt;
   END_STRUCT;
END_TYPE

TYPE "ET_HW_AI"
// stored: IsFailsafeCompliant false
   STRUCT
      HW_AI : Array[0.."ET_AI"] of Int;
   END_STRUCT;
END_TYPE

TYPE "ET_HW_AQ"
// stored: IsFailsafeCompliant false
   STRUCT
      HW_AQ : Array[0.."ET_AQ"] of Int;
   END_STRUCT;
END_TYPE

TYPE "ET_HW_DI"
// stored: IsFailsafeCompliant false
   STRUCT
      HW_DI : Array[0.."ET_DI"] of Bool;
   END_STRUCT;
END_TYPE

TYPE "ET_HW_DQ"
// stored: IsFailsafeCompliant false
   STRUCT
      HW_DQ : Array[0.."ET_DQ"] of Bool;
   END_STRUCT;
END_TYPE

TYPE "PLC_HW_AI"
// stored: IsFailsafeCompliant false
   STRUCT
      HW_AI : Array[0.."PLC_AI"] of Int;
   END_STRUCT;
END_TYPE

TYPE "PLC_HW_AQ"
// stored: IsFailsafeCompliant false
   STRUCT
      HW_AQ : Array[0.."PLC_AQ"] of Int;
   END_STRUCT;
END_TYPE

TYPE "PLC_HW_DI"
// stored: IsFailsafeCompliant false
   STRUCT
      HW_DI : Array[0.."PLC_DI"] of Bool;
   END_STRUCT;
END_TYPE

TYPE "PLC_HW_DQ"
// stored: IsFailsafeCompliant false
   STRUCT
      HW_DQ : Array[0.."PLC_DQ"] of Bool;
   END_STRUCT;
END_TYPE

TYPE "Sequence"
// stored: IsFailsafeCompliant false
   STRUCT
      devOn : Array["MIN_STEP_NUMB".."MAX_STEP_NUMB", "MIN_DEV_NUMB".."MAX_DEV_NUMB"] of Bool;
      delay : Array["MIN_STEP_NUMB".."MAX_STEP_NUMB"] of Int;
   END_STRUCT;
END_TYPE

DATA_BLOCK "dbMain"   // DB2
{ S7_Optimized_Access := 'FALSE' }
VERSION : 0.1
// stored: AutoNumber false, DBAccessibleFromOPCUA true, IsOnlyStoredInLoadMemory false, IsWriteProtectedInAS false
   VAR
      Ack : Bool;
      simUZ : Bool;
      levTW20x : Real;
      levTW140x : Real;
   END_VAR
BEGIN
END_DATA_BLOCK

DATA_BLOCK "dtSetup"   // DB6
{ S7_Optimized_Access := 'FALSE' }
VERSION : 0.1
// stored: AutoNumber true, DBAccessibleFromOPCUA true, IsOnlyStoredInLoadMemory false, IsWriteProtectedInAS false
   VAR RETAIN
      workTW201 : Bool;   // 1-работа, 0-ремонт
      workTW202 : Bool;   // 1-работа, 0-ремонт
      workTW1401 : Bool;   // 1-работа, 0-ремонт
      workTW1402 : Bool;   // 1-работа, 0-ремонт
      selectTW20x : Int;
      selectTW140x : Int;
   END_VAR
BEGIN
END_DATA_BLOCK

DATA_BLOCK "dtAnalogData"   // DB1
{ S7_Optimized_Access := 'FALSE' }
VERSION : 0.1
// stored: AutoNumber true, DBAccessibleFromOPCUA true, IsOnlyStoredInLoadMemory false, IsWriteProtectedInAS false
   VAR
      plc_data : Array[0.."PLC_AI"] of "Ai";
      et_data : Array[0.."ET_AI"] of "Ai";
   END_VAR
BEGIN
   // et_data[0] : aiLT201
   // et_data[1] : aiLT202
   // et_data[2] : aiPT301
   // et_data[3] : aiPT401
   // et_data[4] : aiPT501
   // et_data[5] : aiPT502
   // et_data[6] : aiPT503
   // et_data[7] : aiPT504
   // et_data[8] : aiPT505
   // et_data[9] : aiPT506
   // et_data[10] : aiPT507
   // et_data[11] : aiLT601
   // et_data[12] : aiPT701
   // et_data[13] : aiPT901
   // et_data[14] : aiPT902
   // et_data[15] : aiLT1101
   // et_data[16] : aiPT1201
   // et_data[17] : aiPT1301
   // et_data[18] : aiPT1302
   // et_data[19] : aiLT1401
   // et_data[20] : aiLT1402
   // et_data[21] : aiPT1501
   // et_data[22] : aiPT1701
   // et_data[23] : aiLT1801
   // et_data[24] : aiFM501
   // et_data[25] : aiFM502
   // et_data[26] : aiFM901
   // et_data[27] : aiFM902
   // et_data[28] : aiFM1301
   // et_data[29] : aiFM1302
   // et_data[30] : aiORP801
   // et_data[31] : aiCDI901
   // et_data[32] : aiCDI1301
   // et_data[33] : aiCDI1302
   // et_data[34] : aiCDI1801
END_DATA_BLOCK

DATA_BLOCK "dtDpump"   // DB20
{ S7_Optimized_Access := 'FALSE' }
VERSION : 0.1
// stored: AutoNumber true, DBAccessibleFromOPCUA true, IsOnlyStoredInLoadMemory false, IsWriteProtectedInAS false
   VAR RETAIN
      dp101 : "DPump";
      dp501 : "DPump";
      dp502 : "DPump";
      dp801 : "DPump";
      dp802 : "DPump";
      dp803 : "DPump";
      dp1001 : "DPump";
   END_VAR
BEGIN
END_DATA_BLOCK

DATA_BLOCK "dtPropDpump"   // DB21
{ S7_Optimized_Access := 'FALSE' }
VERSION : 0.1
// stored: AutoNumber true, DBAccessibleFromOPCUA true, IsOnlyStoredInLoadMemory false, IsWriteProtectedInAS false
   VAR RETAIN
      dp101 : "PropDosing";
      dp501 : "PropDosing";
      dp502 : "PropDosing";
      dp801 : "PropDosing";
      dp802 : "PropDosing";
      dp803 : "PropDosing";
      dp1001 : "PropDosing";
   END_VAR
BEGIN
END_DATA_BLOCK

DATA_BLOCK "dtDigitalSensor"   // DB16
{ S7_Optimized_Access := 'FALSE' }
VERSION : 0.1
// stored: AutoNumber true, DBAccessibleFromOPCUA true, IsOnlyStoredInLoadMemory false, IsWriteProtectedInAS false
   VAR RETAIN
      PS901 : "digitalSensor";
      PS902 : "digitalSensor";
      PS1301 : "digitalSensor";
      PS1302 : "digitalSensor";
      FI501 : "digitalSensor";
      FI901 : "digitalSensor";
      FI1301 : "digitalSensor";
   END_VAR
BEGIN
END_DATA_BLOCK

DATA_BLOCK "dbVolumeCounters"   // DB109
{ S7_Optimized_Access := 'FALSE' }
VERSION : 0.1
// stored: AutoNumber true, DBAccessibleFromOPCUA true, IsOnlyStoredInLoadMemory false, IsWriteProtectedInAS false
   VAR RETAIN
      FM201 : "FREQ_COUNTER";   // Витрата вхідної води FM201
      FM501 : "FREQ_COUNTER";   // Витрата вхідної води UF FM501
      FM502 : "FREQ_COUNTER";   // Витрата вхідної води UF FM502
      FM901 : "FREQ_COUNTER";   // Витрата пермеату RO FM901
      FM902 : "FREQ_COUNTER";   // Витрата концентрату RO FM902
      FM1201 : "FREQ_COUNTER";   // Витрата пермеату на споживоча FM1201
      FM1301 : "FREQ_COUNTER";   // Витрата пермеату NF FM1301
      FM1302 : "FREQ_COUNTER";   // Витрата концентрату NF FM1302
      FM1701 : "FREQ_COUNTER";   // Витрата нанофільтрату на споживоча FM1701
      FM1801 : "FREQ_COUNTER";   // Витрата стічних вод FM1801
   END_VAR
BEGIN
END_DATA_BLOCK

DATA_BLOCK "dtParamMDF"   // DB24
{ S7_Optimized_Access := 'FALSE' }
VERSION : 0.1
// stored: AutoNumber true, DBAccessibleFromOPCUA true, IsOnlyStoredInLoadMemory false, IsWriteProtectedInAS false
BEGIN
END_DATA_BLOCK

DATA_BLOCK "dtPID"   // DB8
{ S7_Optimized_Access := 'FALSE' }
VERSION : 0.1
// stored: AutoNumber true, DBAccessibleFromOPCUA true, IsOnlyStoredInLoadMemory false, IsWriteProtectedInAS false
   VAR RETAIN
      pidP30x : "setPID";
      pidP120x { S7_SetPoint := 'True'} : "setPID";
      pidP150x { S7_SetPoint := 'True'} : "setPID";
      pidP901 { S7_SetPoint := 'True'} : "setPID";
      pidP1301 { S7_SetPoint := 'True'} : "setPID";
   END_VAR
BEGIN
END_DATA_BLOCK

DATA_BLOCK "dtPump"   // DB4
{ S7_Optimized_Access := 'FALSE' }
VERSION : 0.1
// stored: AutoNumber true, DBAccessibleFromOPCUA true, IsOnlyStoredInLoadMemory false, IsWriteProtectedInAS false
   VAR RETAIN
      P301 : "Pump";
      P302 { S7_SetPoint := 'True'} : "Pump";
      P1201 { S7_SetPoint := 'True'} : "Pump";
      P1202 { S7_SetPoint := 'True'} : "Pump";
      P1501 { S7_SetPoint := 'True'} : "Pump";
      P1502 { S7_SetPoint := 'True'} : "Pump";
      P701 { S7_SetPoint := 'True'} : "Pump";
      P702 { S7_SetPoint := 'True'} : "Pump";
      P901 { S7_SetPoint := 'True'} : "Pump";
      P1301 { S7_SetPoint := 'True'} : "Pump";
      P2001 { S7_SetPoint := 'True'} : "Pump";
   END_VAR
BEGIN
END_DATA_BLOCK

DATA_BLOCK "dtPumpSetup"   // DB5
{ S7_Optimized_Access := 'FALSE' }
VERSION : 0.1
// stored: AutoNumber true, DBAccessibleFromOPCUA true, IsOnlyStoredInLoadMemory false, IsWriteProtectedInAS false
   VAR RETAIN
      modeP30x : Bool;
      cmStartP30x : Bool;
      selectP30x { S7_SetPoint := 'True'} : Bool;
      freqStopP30x { S7_SetPoint := 'True'} : Real := 31.0;
      delayStopP30x { S7_SetPoint := 'True'} : Real := 5.0;
      presStartP30x { S7_SetPoint := 'True'} : Real := 2.0;
      delayStartP30x { S7_SetPoint := 'True'} : Real := 1.0;
      levTW20xStartP30x { S7_SetPoint := 'True'} : Real := 30.0;
      levTW20xStopP30x { S7_SetPoint := 'True'} : Real := 10.0;
      modeP120x : Bool;
      cmStartP120x : Bool;
      selectP120x { S7_SetPoint := 'True'} : Bool;
      timeNoPulseP120x { S7_SetPoint := 'True'} : Real := 31.0;
      presStartP120x { S7_SetPoint := 'True'} : Real := 2.0;
      delayStartP120x { S7_SetPoint := 'True'} : Real := 1.0;
      levTW11xStartP120x { S7_SetPoint := 'True'} : Real := 30.0;
      levTW11xStopP120x { S7_SetPoint := 'True'} : Real := 10.0;
      modeP150x : Bool;
      cmStartP150x : Bool;
      selectP150x { S7_SetPoint := 'True'} : Bool;
      timeNoPulseP150x { S7_SetPoint := 'True'} : Real := 31.0;
      presStartP150x { S7_SetPoint := 'True'} : Real := 2.0;
      delayStartP150x { S7_SetPoint := 'True'} : Real := 1.0;
      levTW14xStartP150x { S7_SetPoint := 'True'} : Real := 30.0;
      levTW14xStopP150x { S7_SetPoint := 'True'} : Real := 10.0;
      tChangeP30x { S7_SetPoint := 'True'} : Real := 12.0;
      tChangeP120x { S7_SetPoint := 'True'} : Real := 12.0;
      tChangeP150x { S7_SetPoint := 'True'} : Real := 12.0;
      tToChangeP30x : Real;
      tToChangeP120x : Real;
      tToChangeP150x : Real;
      modeP70x : Bool;
      cmP70x : Bool;
      selectP70x : Bool;
      tChangeP70x { S7_SetPoint := 'True'} : Real := 24.0;
      tToChangeP70x : Real;
   END_VAR
BEGIN
END_DATA_BLOCK

DATA_BLOCK "dtUzData"   // DB7
{ S7_Optimized_Access := 'FALSE' }
VERSION : 0.1
// stored: AutoNumber true, DBAccessibleFromOPCUA true, IsOnlyStoredInLoadMemory false, IsWriteProtectedInAS false
   VAR
      UZ30x : "UZ_Data";
      UZ901 { S7_SetPoint := 'True'} : "UZ_Data";
      UZ1301 { S7_SetPoint := 'True'} : "UZ_Data";
      UZ120x { S7_SetPoint := 'True'} : "UZ_Data";
      UZ150x { S7_SetPoint := 'True'} : "UZ_Data";
   END_VAR
BEGIN
END_DATA_BLOCK

DATA_BLOCK "dtParTank"   // DB25
{ S7_Optimized_Access := 'FALSE' }
VERSION : 0.1
// stored: AutoNumber true, DBAccessibleFromOPCUA true, IsOnlyStoredInLoadMemory false, IsWriteProtectedInAS false
   VAR RETAIN
      modeTW1_2 : Int := 2;
   END_VAR
BEGIN
END_DATA_BLOCK

DATA_BLOCK "dtParmUF"   // DB26
{ S7_Optimized_Access := 'FALSE' }
VERSION : 0.1
// stored: AutoNumber true, DBAccessibleFromOPCUA true, IsOnlyStoredInLoadMemory false, IsWriteProtectedInAS false
   VAR RETAIN
      errSettingsLev : Bool;
      filtrationTime : UInt := 10;
      filtrateStartLevUF1 : Real;
      filtrateStopLevUF1 : Real;
      filtrateStartLevUF2 : Real;
      filtrateStopLevUF2 : Real;
      valHDP_ForHW : Real := 1.5;
      minFiltrLevForWash : Real := 50.0;
      delayHDP : UInt := 15;
      maxNumbHW_ByHDP : UInt := 3;
      HW_ToCEB1 : UInt := 3;
      HW_ToCEB2 : UInt := 6;
   END_VAR
BEGIN
END_DATA_BLOCK

DATA_BLOCK "dtUF"   // DB23
{ S7_Optimized_Access := 'FALSE' }
VERSION : 0.1
// stored: AutoNumber true, DBAccessibleFromOPCUA true, IsOnlyStoredInLoadMemory false, IsWriteProtectedInAS false
   VAR RETAIN
      modeUF1 : Bool;
      modeUF2 : Bool;
      cmAuto : Bool;
      flagUF1 : "UF_FLAGS";
      flagUF2 { S7_SetPoint := 'True'} : "UF_FLAGS";
      bUF1 { S7_SetPoint := 'True'} : "UF_COMMANDS";
      bUF2 { S7_SetPoint := 'True'} : "UF_COMMANDS";
      countersUF1 { S7_SetPoint := 'True'} : "UF_COUNTERS";
      countersUF2 { S7_SetPoint := 'True'} : "UF_COUNTERS";
      parUF1 : "UF_PARAMETRS";
      parUF2 { S7_SetPoint := 'True'} : "UF_PARAMETRS";
   END_VAR
BEGIN
END_DATA_BLOCK

DATA_BLOCK "dtUfSeq"   // DB22
{ S7_Optimized_Access := 'FALSE' }
VERSION : 0.1
// stored: AutoNumber true, DBAccessibleFromOPCUA true, IsOnlyStoredInLoadMemory false, IsWriteProtectedInAS false
   VAR RETAIN
      START : "Sequence";
      STOP : "Sequence";
      HW : "Sequence";
      HW_A : "Sequence";
      CEB1 : "Sequence";
      CEB1_A : "Sequence";
      CEB2 : "Sequence";
      CEB2_A : "Sequence";
      SOFT_STOP_UF1 : "Sequence";
      SOFT_STOP_UF2 : "Sequence";
   END_VAR
BEGIN
   START.devOn[1,6] := 1;
   START.devOn[2,1] := 1;
   START.devOn[2,6] := 1;
   START.delay[1..2] := 5;
   STOP.devOn[1,1] := 1;
   STOP.devOn[1,6] := 1;
   STOP.devOn[2,6] := 1;
   STOP.delay[1..2] := 5;
   STOP.delay[3] := 1;
   HW.devOn[1,7] := 1;
   HW.devOn[2,2] := 1;
   HW.devOn[2,7] := 1;
   HW.devOn[3,2..3] := 1;
   HW.devOn[3,7] := 1;
   HW.devOn[4,2..3] := 1;
   HW.devOn[4,5] := 1;
   HW.devOn[4,7] := 1;
   HW.devOn[5,2..3] := 1;
   HW.devOn[5,7] := 1;
   HW.devOn[6,2] := 1;
   HW.devOn[6,7] := 1;
   HW.devOn[7,7] := 1;
   HW.devOn[8,7] := 1;
   HW.devOn[8,10] := 1;
   HW.devOn[9,7] := 1;
   HW.devOn[10,7] := 1;
   HW.devOn[10,9] := 1;
   HW.devOn[11,7] := 1;
   HW.devOn[12,1] := 1;
   HW.devOn[12,7] := 1;
   HW.devOn[13,7] := 1;
   HW.delay[1..3] := 5;
   HW.delay[4] := 10;
   HW.delay[5..7] := 5;
   HW.delay[8] := 10;
   HW.delay[9] := 5;
   HW.delay[10] := 10;
   HW.delay[11] := 5;
   HW.delay[12] := 10;
   HW.delay[13] := 5;
   HW.delay[14] := 1;
   HW_A.devOn[1,7] := 1;
   HW_A.devOn[2,2] := 1;
   HW_A.devOn[2,7] := 1;
   HW_A.devOn[3,2] := 1;
   HW_A.devOn[3,4] := 1;
   HW_A.devOn[3,7] := 1;
   HW_A.devOn[4,2] := 1;
   HW_A.devOn[4,4] := 1;
   HW_A.devOn[4,7] := 1;
   HW_A.devOn[4,11] := 1;
   HW_A.devOn[5,2] := 1;
   HW_A.devOn[5,4] := 1;
   HW_A.devOn[5,7] := 1;
   HW_A.devOn[6,2] := 1;
   HW_A.devOn[6,7] := 1;
   HW_A.devOn[7,7] := 1;
   HW_A.devOn[8,7] := 1;
   HW_A.devOn[8,10] := 1;
   HW_A.devOn[9,7] := 1;
   HW_A.devOn[10,7..8] := 1;
   HW_A.devOn[11,7..9] := 1;
   HW_A.devOn[12,7..8] := 1;
   HW_A.devOn[13,7] := 1;
   HW_A.devOn[14,1] := 1;
   HW_A.devOn[14,7] := 1;
   HW_A.devOn[15,7] := 1;
   HW_A.delay[1..3] := 5;
   HW_A.delay[4] := 10;
   HW_A.delay[5..7] := 5;
   HW_A.delay[8] := 10;
   HW_A.delay[9..10] := 5;
   HW_A.delay[11] := 10;
   HW_A.delay[12..13] := 5;
   HW_A.delay[14] := 10;
   HW_A.delay[15] := 5;
   HW_A.delay[16] := 1;
   CEB1.devOn[1,7] := 1;
   CEB1.devOn[2,7..8] := 1;
   CEB1.devOn[3,2] := 1;
   CEB1.devOn[3,7..8] := 1;
   CEB1.devOn[4,2..3] := 1;
   CEB1.devOn[4,7..8] := 1;
   CEB1.devOn[5,2..3] := 1;
   CEB1.devOn[5,5] := 1;
   CEB1.devOn[5,7..8] := 1;
   CEB1.devOn[5,13] := 1;
   CEB1.devOn[6,2..3] := 1;
   CEB1.devOn[6,5] := 1;
   CEB1.devOn[6,7] := 1;
   CEB1.devOn[6,13] := 1;
   CEB1.devOn[7,2..3] := 1;
   CEB1.devOn[7,7] := 1;
   CEB1.devOn[8,2] := 1;
   CEB1.devOn[8,7] := 1;
   CEB1.devOn[9,7] := 1;
   CEB1.devOn[10,7] := 1;
   CEB1.devOn[10,10] := 1;
   CEB1.devOn[11,7] := 1;
   CEB1.devOn[12,7] := 1;
   CEB1.devOn[12,9] := 1;
   CEB1.devOn[13,7..9] := 1;
   CEB1.devOn[14,7] := 1;
   CEB1.devOn[14,9] := 1;
   CEB1.devOn[15,7] := 1;
   CEB1.devOn[16,2] := 1;
   CEB1.devOn[16,7] := 1;
   CEB1.devOn[17,2..3] := 1;
   CEB1.devOn[17,7] := 1;
   CEB1.devOn[18,2..3] := 1;
   CEB1.devOn[18,5] := 1;
   CEB1.devOn[18,7] := 1;
   CEB1.devOn[19,2..3] := 1;
   CEB1.devOn[19,7] := 1;
   CEB1.devOn[20,2] := 1;
   CEB1.devOn[20,7] := 1;
   CEB1.devOn[21,7] := 1;
   CEB1.devOn[22,7] := 1;
   CEB1.devOn[22,10] := 1;
   CEB1.devOn[23,7] := 1;
   CEB1.devOn[24,7] := 1;
   CEB1.devOn[24,9] := 1;
   CEB1.devOn[25,7..9] := 1;
   CEB1.devOn[26,7] := 1;
   CEB1.devOn[26,9] := 1;
   CEB1.devOn[27,7] := 1;
   CEB1.devOn[28,2] := 1;
   CEB1.devOn[28,7] := 1;
   CEB1.devOn[29,2..3] := 1;
   CEB1.devOn[29,7] := 1;
   CEB1.devOn[30,2..3] := 1;
   CEB1.devOn[30,5] := 1;
   CEB1.devOn[30,7] := 1;
   CEB1.devOn[31,2..3] := 1;
   CEB1.devOn[31,8] := 1;
   CEB1.devOn[32,2] := 1;
   CEB1.devOn[32,7] := 1;
   CEB1.devOn[33,7] := 1;
   CEB1.devOn[34,7] := 1;
   CEB1.devOn[34,10] := 1;
   CEB1.devOn[35,7] := 1;
   CEB1.devOn[36,7] := 1;
   CEB1.devOn[36,9] := 1;
   CEB1.devOn[37,7..9] := 1;
   CEB1.devOn[38,7] := 1;
   CEB1.devOn[38,9] := 1;
   CEB1.devOn[39,7] := 1;
   CEB1.devOn[40,1] := 1;
   CEB1.devOn[40,7] := 1;
   CEB1.devOn[41,7] := 1;
   CEB1.delay[1..4] := 5;
   CEB1.delay[5] := 10;
   CEB1.delay[6..8] := 5;
   CEB1.delay[9..10] := 10;
   CEB1.delay[11..12] := 5;
   CEB1.delay[13] := 10;
   CEB1.delay[14..17] := 5;
   CEB1.delay[18] := 10;
   CEB1.delay[19..21] := 5;
   CEB1.delay[22] := 10;
   CEB1.delay[23..24] := 5;
   CEB1.delay[25] := 10;
   CEB1.delay[26..29] := 5;
   CEB1.delay[30] := 10;
   CEB1.delay[31..33] := 5;
   CEB1.delay[34] := 10;
   CEB1.delay[35..36] := 5;
   CEB1.delay[37] := 10;
   CEB1.delay[38..39] := 5;
   CEB1.delay[40] := 10;
   CEB1.delay[41] := 5;
   CEB1.delay[42] := 1;
   CEB1_A.devOn[1,1..6] := false;
   CEB1_A.devOn[1,7] := 1;
   CEB1_A.devOn[1,8..16] := false;
   CEB1_A.devOn[2,1..6] := false;
   CEB1_A.devOn[2,7..8] := 1;
   CEB1_A.devOn[2,9..16] := false;
   CEB1_A.devOn[3,1] := false;
   CEB1_A.devOn[3,2] := 1;
   CEB1_A.devOn[3,3..6] := false;
   CEB1_A.devOn[3,7..8] := 1;
   CEB1_A.devOn[3,9..16] := false;
   CEB1_A.devOn[4,1] := false;
   CEB1_A.devOn[4,2] := 1;
   CEB1_A.devOn[4,4] := 1;
   CEB1_A.devOn[4,5..6] := false;
   CEB1_A.devOn[4,7..8] := 1;
   CEB1_A.devOn[4,9..16] := false;
   CEB1_A.devOn[5,1] := false;
   CEB1_A.devOn[5,2] := 1;
   CEB1_A.devOn[5,4] := 1;
   CEB1_A.devOn[5,6] := false;
   CEB1_A.devOn[5,7..8] := 1;
   CEB1_A.devOn[5,9..10] := false;
   CEB1_A.devOn[5,11] := 1;
   CEB1_A.devOn[5,12] := false;
   CEB1_A.devOn[5,13] := 1;
   CEB1_A.devOn[5,14..16] := false;
   CEB1_A.devOn[6,1] := false;
   CEB1_A.devOn[6,2] := 1;
   CEB1_A.devOn[6,4] := 1;
   CEB1_A.devOn[6,6] := false;
   CEB1_A.devOn[6,7] := 1;
   CEB1_A.devOn[6,8..10] := false;
   CEB1_A.devOn[6,11] := 1;
   CEB1_A.devOn[6,12] := false;
   CEB1_A.devOn[6,13] := 1;
   CEB1_A.devOn[6,14..16] := false;
   CEB1_A.devOn[7,1] := false;
   CEB1_A.devOn[7,2] := 1;
   CEB1_A.devOn[7,4] := 1;
   CEB1_A.devOn[7,5..6] := false;
   CEB1_A.devOn[7,7] := 1;
   CEB1_A.devOn[7,8..16] := false;
   CEB1_A.devOn[8,1] := false;
   CEB1_A.devOn[8,2] := 1;
   CEB1_A.devOn[8,3..6] := false;
   CEB1_A.devOn[8,7] := 1;
   CEB1_A.devOn[8,8..16] := false;
   CEB1_A.devOn[9,1..6] := false;
   CEB1_A.devOn[9,7] := 1;
   CEB1_A.devOn[9,8..16] := false;
   CEB1_A.devOn[10,1..6] := false;
   CEB1_A.devOn[10,7] := 1;
   CEB1_A.devOn[10,8..9] := false;
   CEB1_A.devOn[10,10] := 1;
   CEB1_A.devOn[10,11..16] := false;
   CEB1_A.devOn[11,1..6] := false;
   CEB1_A.devOn[11,7] := 1;
   CEB1_A.devOn[11,8..16] := false;
   CEB1_A.devOn[12,1..6] := false;
   CEB1_A.devOn[12,7] := 1;
   CEB1_A.devOn[12,8] := false;
   CEB1_A.devOn[12,9] := 1;
   CEB1_A.devOn[12,10..16] := false;
   CEB1_A.devOn[13,1..6] := false;
   CEB1_A.devOn[13,7..9] := 1;
   CEB1_A.devOn[13,10..16] := false;
   CEB1_A.devOn[14,1..6] := false;
   CEB1_A.devOn[14,7] := 1;
   CEB1_A.devOn[14,8] := false;
   CEB1_A.devOn[14,9] := 1;
   CEB1_A.devOn[14,10..16] := false;
   CEB1_A.devOn[15,1..6] := false;
   CEB1_A.devOn[15,7] := 1;
   CEB1_A.devOn[15,8..16] := false;
   CEB1_A.devOn[16,1] := false;
   CEB1_A.devOn[16,2] := 1;
   CEB1_A.devOn[16,3..6] := false;
   CEB1_A.devOn[16,7] := 1;
   CEB1_A.devOn[16,8..16] := false;
   CEB1_A.devOn[17,1] := false;
   CEB1_A.devOn[17,2] := 1;
   CEB1_A.devOn[17,4] := 1;
   CEB1_A.devOn[17,5..6] := false;
   CEB1_A.devOn[17,7] := 1;
   CEB1_A.devOn[17,8..16] := false;
   CEB1_A.devOn[18,1] := false;
   CEB1_A.devOn[18,2] := 1;
   CEB1_A.devOn[18,4] := 1;
   CEB1_A.devOn[18,6] := false;
   CEB1_A.devOn[18,7] := 1;
   CEB1_A.devOn[18,8..10] := false;
   CEB1_A.devOn[18,11] := 1;
   CEB1_A.devOn[18,12..16] := false;
   CEB1_A.devOn[19,1] := false;
   CEB1_A.devOn[19,2] := 1;
   CEB1_A.devOn[19,4] := 1;
   CEB1_A.devOn[19,5..6] := false;
   CEB1_A.devOn[19,7] := 1;
   CEB1_A.devOn[19,8..16] := false;
   CEB1_A.devOn[20,1] := false;
   CEB1_A.devOn[20,2] := 1;
   CEB1_A.devOn[20,3..6] := false;
   CEB1_A.devOn[20,7] := 1;
   CEB1_A.devOn[20,8..16] := false;
   CEB1_A.devOn[21,1..6] := false;
   CEB1_A.devOn[21,7] := 1;
   CEB1_A.devOn[21,8..16] := false;
   CEB1_A.devOn[22,1..6] := false;
   CEB1_A.devOn[22,7] := 1;
   CEB1_A.devOn[22,8..9] := false;
   CEB1_A.devOn[22,10] := 1;
   CEB1_A.devOn[22,11..16] := false;
   CEB1_A.devOn[23,1..6] := false;
   CEB1_A.devOn[23,7] := 1;
   CEB1_A.devOn[23,8..16] := false;
   CEB1_A.devOn[24,1..6] := false;
   CEB1_A.devOn[24,7] := 1;
   CEB1_A.devOn[24,8] := false;
   CEB1_A.devOn[24,9] := 1;
   CEB1_A.devOn[24,10..16] := false;
   CEB1_A.devOn[25,1..6] := false;
   CEB1_A.devOn[25,7..9] := 1;
   CEB1_A.devOn[25,10..16] := false;
   CEB1_A.devOn[26,1..6] := false;
   CEB1_A.devOn[26,7] := 1;
   CEB1_A.devOn[26,8] := false;
   CEB1_A.devOn[26,9] := 1;
   CEB1_A.devOn[26,10..16] := false;
   CEB1_A.devOn[27,1..6] := false;
   CEB1_A.devOn[27,7] := 1;
   CEB1_A.devOn[27,8..16] := false;
   CEB1_A.devOn[28,1] := false;
   CEB1_A.devOn[28,2] := 1;
   CEB1_A.devOn[28,3..6] := false;
   CEB1_A.devOn[28,7] := 1;
   CEB1_A.devOn[28,8..16] := false;
   CEB1_A.devOn[29,1] := false;
   CEB1_A.devOn[29,2] := 1;
   CEB1_A.devOn[29,3] := false;
   CEB1_A.devOn[29,4] := 1;
   CEB1_A.devOn[29,5..6] := false;
   CEB1_A.devOn[29,7] := 1;
   CEB1_A.devOn[29,8..16] := false;
   CEB1_A.devOn[30,1] := false;
   CEB1_A.devOn[30,2] := 1;
   CEB1_A.devOn[30,3] := false;
   CEB1_A.devOn[30,4] := 1;
   CEB1_A.devOn[30,5..6] := false;
   CEB1_A.devOn[30,7] := 1;
   CEB1_A.devOn[30,8..10] := false;
   CEB1_A.devOn[30,11] := 1;
   CEB1_A.devOn[30,12..16] := false;
   CEB1_A.devOn[31,1] := false;
   CEB1_A.devOn[31,2] := 1;
   CEB1_A.devOn[31,3] := false;
   CEB1_A.devOn[31,4] := 1;
   CEB1_A.devOn[31,5..6] := false;
   CEB1_A.devOn[31,7] := 1;
   CEB1_A.devOn[31,8..16] := false;
   CEB1_A.devOn[32,1] := false;
   CEB1_A.devOn[32,2] := 1;
   CEB1_A.devOn[32,3..6] := false;
   CEB1_A.devOn[32,7] := 1;
   CEB1_A.devOn[32,8..16] := false;
   CEB1_A.devOn[33,1..6] := false;
   CEB1_A.devOn[33,7] := 1;
   CEB1_A.devOn[33,8..16] := false;
   CEB1_A.devOn[34,1..6] := false;
   CEB1_A.devOn[34,7] := 1;
   CEB1_A.devOn[34,8..9] := false;
   CEB1_A.devOn[34,10] := 1;
   CEB1_A.devOn[34,11..16] := false;
   CEB1_A.devOn[35,1..6] := false;
   CEB1_A.devOn[35,7] := 1;
   CEB1_A.devOn[35,8..16] := false;
   CEB1_A.devOn[36,1..6] := false;
   CEB1_A.devOn[36,7] := 1;
   CEB1_A.devOn[36,8] := false;
   CEB1_A.devOn[36,9] := 1;
   CEB1_A.devOn[36,10..16] := false;
   CEB1_A.devOn[37,1..6] := false;
   CEB1_A.devOn[37,7..9] := 1;
   CEB1_A.devOn[37,10..16] := false;
   CEB1_A.devOn[38,1..6] := false;
   CEB1_A.devOn[38,7] := 1;
   CEB1_A.devOn[38,8] := false;
   CEB1_A.devOn[38,9] := 1;
   CEB1_A.devOn[38,10..16] := false;
   CEB1_A.devOn[39,1..6] := false;
   CEB1_A.devOn[39,7] := 1;
   CEB1_A.devOn[39,8..16] := false;
   CEB1_A.devOn[40,1] := 1;
   CEB1_A.devOn[40,2..6] := false;
   CEB1_A.devOn[40,7] := 1;
   CEB1_A.devOn[40,8..16] := false;
   CEB1_A.devOn[41,1..6] := false;
   CEB1_A.devOn[41,7] := 1;
   CEB1_A.devOn[41,8..16] := false;
   CEB1_A.delay[1..4] := 5;
   CEB1_A.delay[5] := 10;
   CEB1_A.delay[6..8] := 5;
   CEB1_A.delay[9..10] := 10;
   CEB1_A.delay[11..12] := 5;
   CEB1_A.delay[13] := 10;
   CEB1_A.delay[14..17] := 5;
   CEB1_A.delay[18] := 10;
   CEB1_A.delay[19..21] := 5;
   CEB1_A.delay[22] := 10;
   CEB1_A.delay[23..24] := 5;
   CEB1_A.delay[25] := 10;
   CEB1_A.delay[26..29] := 5;
   CEB1_A.delay[30] := 10;
   CEB1_A.delay[31..33] := 5;
   CEB1_A.delay[34] := 10;
   CEB1_A.delay[35..36] := 5;
   CEB1_A.delay[37] := 10;
   CEB1_A.delay[38..39] := 5;
   CEB1_A.delay[40] := 10;
   CEB1_A.delay[41] := 5;
   CEB1_A.delay[42] := 1;
   CEB2.devOn[1,1..6] := false;
   CEB2.devOn[1,7] := 1;
   CEB2.devOn[1,8..16] := false;
   CEB2.devOn[2,1..6] := false;
   CEB2.devOn[2,7..8] := 1;
   CEB2.devOn[2,9..16] := false;
   CEB2.devOn[3,1] := false;
   CEB2.devOn[3,2] := 1;
   CEB2.devOn[3,3..6] := false;
   CEB2.devOn[3,7..8] := 1;
   CEB2.devOn[3,9..16] := false;
   CEB2.devOn[4,1] := false;
   CEB2.devOn[4,2..3] := 1;
   CEB2.devOn[4,4..6] := false;
   CEB2.devOn[4,7..8] := 1;
   CEB2.devOn[4,9..16] := false;
   CEB2.devOn[5,1] := false;
   CEB2.devOn[5,2..3] := 1;
   CEB2.devOn[5,4] := false;
   CEB2.devOn[5,5] := 1;
   CEB2.devOn[5,6] := false;
   CEB2.devOn[5,7..8] := 1;
   CEB2.devOn[5,9..11] := false;
   CEB2.devOn[5,12] := 1;
   CEB2.devOn[5,14..16] := false;
   CEB2.devOn[6,1] := false;
   CEB2.devOn[6,2..3] := 1;
   CEB2.devOn[6,4] := false;
   CEB2.devOn[6,5] := 1;
   CEB2.devOn[6,6] := false;
   CEB2.devOn[6,7] := 1;
   CEB2.devOn[6,8..11] := false;
   CEB2.devOn[6,12] := 1;
   CEB2.devOn[6,14..16] := false;
   CEB2.devOn[7,1] := false;
   CEB2.devOn[7,2..3] := 1;
   CEB2.devOn[7,4..6] := false;
   CEB2.devOn[7,7] := 1;
   CEB2.devOn[7,8..16] := false;
   CEB2.devOn[8,1] := false;
   CEB2.devOn[8,2] := 1;
   CEB2.devOn[8,3..6] := false;
   CEB2.devOn[8,7] := 1;
   CEB2.devOn[8,8..16] := false;
   CEB2.devOn[9,1..6] := false;
   CEB2.devOn[9,7] := 1;
   CEB2.devOn[9,8..16] := false;
   CEB2.devOn[10,1..6] := false;
   CEB2.devOn[10,7] := 1;
   CEB2.devOn[10,8..9] := false;
   CEB2.devOn[10,10] := 1;
   CEB2.devOn[10,11..16] := false;
   CEB2.devOn[11,1..6] := false;
   CEB2.devOn[11,7] := 1;
   CEB2.devOn[11,8..16] := false;
   CEB2.devOn[12,1..6] := false;
   CEB2.devOn[12,7] := 1;
   CEB2.devOn[12,8] := false;
   CEB2.devOn[12,9] := 1;
   CEB2.devOn[12,10..16] := false;
   CEB2.devOn[13,1..6] := false;
   CEB2.devOn[13,7..9] := 1;
   CEB2.devOn[13,10..16] := false;
   CEB2.devOn[14,1..6] := false;
   CEB2.devOn[14,7] := 1;
   CEB2.devOn[14,8] := false;
   CEB2.devOn[14,9] := 1;
   CEB2.devOn[14,10..16] := false;
   CEB2.devOn[15,1..6] := false;
   CEB2.devOn[15,7] := 1;
   CEB2.devOn[15,8..16] := false;
   CEB2.devOn[16,1] := false;
   CEB2.devOn[16,2] := 1;
   CEB2.devOn[16,3..6] := false;
   CEB2.devOn[16,7] := 1;
   CEB2.devOn[16,8..16] := false;
   CEB2.devOn[17,1] := false;
   CEB2.devOn[17,2..3] := 1;
   CEB2.devOn[17,4..6] := false;
   CEB2.devOn[17,7] := 1;
   CEB2.devOn[17,8..16] := false;
   CEB2.devOn[18,1] := false;
   CEB2.devOn[18,2..3] := 1;
   CEB2.devOn[18,4] := false;
   CEB2.devOn[18,5] := 1;
   CEB2.devOn[18,6] := false;
   CEB2.devOn[18,7] := 1;
   CEB2.devOn[18,8..16] := false;
   CEB2.devOn[19,1] := false;
   CEB2.devOn[19,2..3] := 1;
   CEB2.devOn[19,4..6] := false;
   CEB2.devOn[19,7] := 1;
   CEB2.devOn[19,8..16] := false;
   CEB2.devOn[20,1] := false;
   CEB2.devOn[20,2] := 1;
   CEB2.devOn[20,3..6] := false;
   CEB2.devOn[20,7] := 1;
   CEB2.devOn[20,8..16] := false;
   CEB2.devOn[21,1..6] := false;
   CEB2.devOn[21,7] := 1;
   CEB2.devOn[21,8..16] := false;
   CEB2.devOn[22,1..6] := false;
   CEB2.devOn[22,7] := 1;
   CEB2.devOn[22,8..9] := false;
   CEB2.devOn[22,10] := 1;
   CEB2.devOn[22,11..16] := false;
   CEB2.devOn[23,1..6] := false;
   CEB2.devOn[23,7] := 1;
   CEB2.devOn[23,8..16] := false;
   CEB2.devOn[24,1..6] := false;
   CEB2.devOn[24,7] := 1;
   CEB2.devOn[24,8] := false;
   CEB2.devOn[24,9] := 1;
   CEB2.devOn[24,10..16] := false;
   CEB2.devOn[25,1..6] := false;
   CEB2.devOn[25,7..9] := 1;
   CEB2.devOn[25,10..16] := false;
   CEB2.devOn[26,1..6] := false;
   CEB2.devOn[26,7] := 1;
   CEB2.devOn[26,8] := false;
   CEB2.devOn[26,9] := 1;
   CEB2.devOn[26,10..16] := false;
   CEB2.devOn[27,1..6] := false;
   CEB2.devOn[27,7] := 1;
   CEB2.devOn[27,8..16] := false;
   CEB2.devOn[28,1] := false;
   CEB2.devOn[28,2] := 1;
   CEB2.devOn[28,3..6] := false;
   CEB2.devOn[28,7] := 1;
   CEB2.devOn[28,8..16] := false;
   CEB2.devOn[29,1] := false;
   CEB2.devOn[29,2..3] := 1;
   CEB2.devOn[29,4..6] := false;
   CEB2.devOn[29,7] := 1;
   CEB2.devOn[29,8..16] := false;
   CEB2.devOn[30,1] := false;
   CEB2.devOn[30,2..3] := 1;
   CEB2.devOn[30,4] := false;
   CEB2.devOn[30,5] := 1;
   CEB2.devOn[30,6] := false;
   CEB2.devOn[30,7] := 1;
   CEB2.devOn[30,8..16] := false;
   CEB2.devOn[31,1] := false;
   CEB2.devOn[31,2..3] := 1;
   CEB2.devOn[31,4..7] := false;
   CEB2.devOn[31,8] := 1;
   CEB2.devOn[31,9..16] := false;
   CEB2.devOn[32,1] := false;
   CEB2.devOn[32,2] := 1;
   CEB2.devOn[32,3..6] := false;
   CEB2.devOn[32,7] := 1;
   CEB2.devOn[32,8..16] := false;
   CEB2.devOn[33,1..6] := false;
   CEB2.devOn[33,7] := 1;
   CEB2.devOn[33,8..16] := false;
   CEB2.devOn[34,1..6] := false;
   CEB2.devOn[34,7] := 1;
   CEB2.devOn[34,8..9] := false;
   CEB2.devOn[34,10] := 1;
   CEB2.devOn[34,11..16] := false;
   CEB2.devOn[35,1..6] := false;
   CEB2.devOn[35,7] := 1;
   CEB2.devOn[35,8..16] := false;
   CEB2.devOn[36,1..6] := false;
   CEB2.devOn[36,7] := 1;
   CEB2.devOn[36,8] := false;
   CEB2.devOn[36,9] := 1;
   CEB2.devOn[36,10..16] := false;
   CEB2.devOn[37,1..6] := false;
   CEB2.devOn[37,7..9] := 1;
   CEB2.devOn[37,10..16] := false;
   CEB2.devOn[38,1..6] := false;
   CEB2.devOn[38,7] := 1;
   CEB2.devOn[38,8] := false;
   CEB2.devOn[38,9] := 1;
   CEB2.devOn[38,10..16] := false;
   CEB2.devOn[39,1..6] := false;
   CEB2.devOn[39,7] := 1;
   CEB2.devOn[39,8..16] := false;
   CEB2.devOn[40,1] := 1;
   CEB2.devOn[40,2..6] := false;
   CEB2.devOn[40,7] := 1;
   CEB2.devOn[40,8..16] := false;
   CEB2.devOn[41,1..6] := false;
   CEB2.devOn[41,7] := 1;
   CEB2.devOn[41,8..16] := false;
   CEB2.delay[1..4] := 5;
   CEB2.delay[5] := 10;
   CEB2.delay[6..8] := 5;
   CEB2.delay[9..10] := 10;
   CEB2.delay[11..12] := 5;
   CEB2.delay[13] := 10;
   CEB2.delay[14..17] := 5;
   CEB2.delay[18] := 10;
   CEB2.delay[19..21] := 5;
   CEB2.delay[22] := 10;
   CEB2.delay[23..24] := 5;
   CEB2.delay[25] := 10;
   CEB2.delay[26..29] := 5;
   CEB2.delay[30] := 10;
   CEB2.delay[31..33] := 5;
   CEB2.delay[34] := 10;
   CEB2.delay[35..36] := 5;
   CEB2.delay[37] := 10;
   CEB2.delay[38..39] := 5;
   CEB2.delay[40] := 10;
   CEB2.delay[41] := 5;
   CEB2.delay[42] := 1;
   CEB2_A.devOn[1,1..6] := false;
   CEB2_A.devOn[1,7] := 1;
   CEB2_A.devOn[1,8..16] := false;
   CEB2_A.devOn[2,1..6] := false;
   CEB2_A.devOn[2,7..8] := 1;
   CEB2_A.devOn[2,9..16] := false;
   CEB2_A.devOn[3,1] := false;
   CEB2_A.devOn[3,2] := 1;
   CEB2_A.devOn[3,3..6] := false;
   CEB2_A.devOn[3,7..8] := 1;
   CEB2_A.devOn[3,9..16] := false;
   CEB2_A.devOn[4,1] := false;
   CEB2_A.devOn[4,2] := 1;
   CEB2_A.devOn[4,3] := false;
   CEB2_A.devOn[4,4] := 1;
   CEB2_A.devOn[4,5..6] := false;
   CEB2_A.devOn[4,7..8] := 1;
   CEB2_A.devOn[4,9..16] := false;
   CEB2_A.devOn[5,1] := false;
   CEB2_A.devOn[5,2] := 1;
   CEB2_A.devOn[5,3] := false;
   CEB2_A.devOn[5,4] := 1;
   CEB2_A.devOn[5,5..6] := false;
   CEB2_A.devOn[5,7..8] := 1;
   CEB2_A.devOn[5,9..10] := false;
   CEB2_A.devOn[5,11..12] := 1;
   CEB2_A.devOn[5,14..16] := false;
   CEB2_A.devOn[6,1] := false;
   CEB2_A.devOn[6,2] := 1;
   CEB2_A.devOn[6,3] := false;
   CEB2_A.devOn[6,4] := 1;
   CEB2_A.devOn[6,5..6] := false;
   CEB2_A.devOn[6,7] := 1;
   CEB2_A.devOn[6,8..10] := false;
   CEB2_A.devOn[6,11..12] := 1;
   CEB2_A.devOn[6,14..16] := false;
   CEB2_A.devOn[7,1] := false;
   CEB2_A.devOn[7,2] := 1;
   CEB2_A.devOn[7,3] := false;
   CEB2_A.devOn[7,4] := 1;
   CEB2_A.devOn[7,5..6] := false;
   CEB2_A.devOn[7,7] := 1;
   CEB2_A.devOn[7,8..16] := false;
   CEB2_A.devOn[8,1] := false;
   CEB2_A.devOn[8,2] := 1;
   CEB2_A.devOn[8,3..6] := false;
   CEB2_A.devOn[8,7] := 1;
   CEB2_A.devOn[8,8..16] := false;
   CEB2_A.devOn[9,1..6] := false;
   CEB2_A.devOn[9,7] := 1;
   CEB2_A.devOn[9,8..16] := false;
   CEB2_A.devOn[10,1..6] := false;
   CEB2_A.devOn[10,7] := 1;
   CEB2_A.devOn[10,8..9] := false;
   CEB2_A.devOn[10,10] := 1;
   CEB2_A.devOn[10,11..16] := false;
   CEB2_A.devOn[11,1..6] := false;
   CEB2_A.devOn[11,7] := 1;
   CEB2_A.devOn[11,8..16] := false;
   CEB2_A.devOn[12,1..6] := false;
   CEB2_A.devOn[12,7] := 1;
   CEB2_A.devOn[12,8] := false;
   CEB2_A.devOn[12,9] := 1;
   CEB2_A.devOn[12,10..16] := false;
   CEB2_A.devOn[13,1..6] := false;
   CEB2_A.devOn[13,7..9] := 1;
   CEB2_A.devOn[13,10..16] := false;
   CEB2_A.devOn[14,1..6] := false;
   CEB2_A.devOn[14,7] := 1;
   CEB2_A.devOn[14,8] := false;
   CEB2_A.devOn[14,9] := 1;
   CEB2_A.devOn[14,10..16] := false;
   CEB2_A.devOn[15,1..6] := false;
   CEB2_A.devOn[15,7] := 1;
   CEB2_A.devOn[15,8..16] := false;
   CEB2_A.devOn[16,1] := false;
   CEB2_A.devOn[16,2] := 1;
   CEB2_A.devOn[16,3..6] := false;
   CEB2_A.devOn[16,7] := 1;
   CEB2_A.devOn[16,8..16] := false;
   CEB2_A.devOn[17,1] := false;
   CEB2_A.devOn[17,2] := 1;
   CEB2_A.devOn[17,3] := false;
   CEB2_A.devOn[17,4] := 1;
   CEB2_A.devOn[17,5..6] := false;
   CEB2_A.devOn[17,7] := 1;
   CEB2_A.devOn[17,8..16] := false;
   CEB2_A.devOn[18,1] := false;
   CEB2_A.devOn[18,2] := 1;
   CEB2_A.devOn[18,3] := false;
   CEB2_A.devOn[18,4] := 1;
   CEB2_A.devOn[18,5..6] := false;
   CEB2_A.devOn[18,7] := 1;
   CEB2_A.devOn[18,8..10] := false;
   CEB2_A.devOn[18,11] := 1;
   CEB2_A.devOn[18,12..16] := false;
   CEB2_A.devOn[19,1] := false;
   CEB2_A.devOn[19,2] := 1;
   CEB2_A.devOn[19,3] := false;
   CEB2_A.devOn[19,4] := 1;
   CEB2_A.devOn[19,5..6] := false;
   CEB2_A.devOn[19,7] := 1;
   CEB2_A.devOn[19,8..16] := false;
   CEB2_A.devOn[20,1] := false;
   CEB2_A.devOn[20,2] := 1;
   CEB2_A.devOn[20,3..6] := false;
   CEB2_A.devOn[20,7] := 1;
   CEB2_A.devOn[20,8..16] := false;
   CEB2_A.devOn[21,1..6] := false;
   CEB2_A.devOn[21,7] := 1;
   CEB2_A.devOn[21,8..16] := false;
   CEB2_A.devOn[22,1..6] := false;
   CEB2_A.devOn[22,7] := 1;
   CEB2_A.devOn[22,8..9] := false;
   CEB2_A.devOn[22,10] := 1;
   CEB2_A.devOn[22,11..16] := false;
   CEB2_A.devOn[23,1..6] := false;
   CEB2_A.devOn[23,7] := 1;
   CEB2_A.devOn[23,8..16] := false;
   CEB2_A.devOn[24,1..6] := false;
   CEB2_A.devOn[24,7] := 1;
   CEB2_A.devOn[24,8] := false;
   CEB2_A.devOn[24,9] := 1;
   CEB2_A.devOn[24,10..16] := false;
   CEB2_A.devOn[25,1..6] := false;
   CEB2_A.devOn[25,7..9] := 1;
   CEB2_A.devOn[25,10..16] := false;
   CEB2_A.devOn[26,1..6] := false;
   CEB2_A.devOn[26,7] := 1;
   CEB2_A.devOn[26,8] := false;
   CEB2_A.devOn[26,9] := 1;
   CEB2_A.devOn[26,10..16] := false;
   CEB2_A.devOn[27,1..6] := false;
   CEB2_A.devOn[27,7] := 1;
   CEB2_A.devOn[27,8..16] := false;
   CEB2_A.devOn[28,1] := false;
   CEB2_A.devOn[28,2] := 1;
   CEB2_A.devOn[28,3..6] := false;
   CEB2_A.devOn[28,7] := 1;
   CEB2_A.devOn[28,8..16] := false;
   CEB2_A.devOn[29,1] := false;
   CEB2_A.devOn[29,2] := 1;
   CEB2_A.devOn[29,3] := false;
   CEB2_A.devOn[29,4] := 1;
   CEB2_A.devOn[29,5..6] := false;
   CEB2_A.devOn[29,7] := 1;
   CEB2_A.devOn[29,8..16] := false;
   CEB2_A.devOn[30,1] := false;
   CEB2_A.devOn[30,2] := 1;
   CEB2_A.devOn[30,3] := false;
   CEB2_A.devOn[30,4] := 1;
   CEB2_A.devOn[30,5..6] := false;
   CEB2_A.devOn[30,7] := 1;
   CEB2_A.devOn[30,8..10] := false;
   CEB2_A.devOn[30,11] := 1;
   CEB2_A.devOn[30,12..16] := false;
   CEB2_A.devOn[31,1] := false;
   CEB2_A.devOn[31,2] := 1;
   CEB2_A.devOn[31,3] := false;
   CEB2_A.devOn[31,4] := 1;
   CEB2_A.devOn[31,5..6] := false;
   CEB2_A.devOn[31,7] := 1;
   CEB2_A.devOn[31,8..16] := false;
   CEB2_A.devOn[32,1] := false;
   CEB2_A.devOn[32,2] := 1;
   CEB2_A.devOn[32,3..6] := false;
   CEB2_A.devOn[32,7] := 1;
   CEB2_A.devOn[32,8..16] := false;
   CEB2_A.devOn[33,1..6] := false;
   CEB2_A.devOn[33,7] := 1;
   CEB2_A.devOn[33,8..16] := false;
   CEB2_A.devOn[34,1..6] := false;
   CEB2_A.devOn[34,7] := 1;
   CEB2_A.devOn[34,8..9] := false;
   CEB2_A.devOn[34,10] := 1;
   CEB2_A.devOn[34,11..16] := false;
   CEB2_A.devOn[35,1..6] := false;
   CEB2_A.devOn[35,7] := 1;
   CEB2_A.devOn[35,8..16] := false;
   CEB2_A.devOn[36,1..6] := false;
   CEB2_A.devOn[36,7] := 1;
   CEB2_A.devOn[36,8] := false;
   CEB2_A.devOn[36,9] := 1;
   CEB2_A.devOn[36,10..16] := false;
   CEB2_A.devOn[37,1..6] := false;
   CEB2_A.devOn[37,7..9] := 1;
   CEB2_A.devOn[37,10..16] := false;
   CEB2_A.devOn[38,1..6] := false;
   CEB2_A.devOn[38,7] := 1;
   CEB2_A.devOn[38,8] := false;
   CEB2_A.devOn[38,9] := 1;
   CEB2_A.devOn[38,10..16] := false;
   CEB2_A.devOn[39,1..6] := false;
   CEB2_A.devOn[39,7] := 1;
   CEB2_A.devOn[39,8..16] := false;
   CEB2_A.devOn[40,1] := 1;
   CEB2_A.devOn[40,2..6] := false;
   CEB2_A.devOn[40,7] := 1;
   CEB2_A.devOn[40,8..16] := false;
   CEB2_A.devOn[41,1..6] := false;
   CEB2_A.devOn[41,7] := 1;
   CEB2_A.devOn[41,8..16] := false;
   CEB2_A.delay[1..4] := 5;
   CEB2_A.delay[5] := 10;
   CEB2_A.delay[6..8] := 5;
   CEB2_A.delay[9..10] := 10;
   CEB2_A.delay[11..12] := 5;
   CEB2_A.delay[13] := 10;
   CEB2_A.delay[14..17] := 5;
   CEB2_A.delay[18] := 10;
   CEB2_A.delay[19..21] := 5;
   CEB2_A.delay[22] := 10;
   CEB2_A.delay[23..24] := 5;
   CEB2_A.delay[25] := 10;
   CEB2_A.delay[26..29] := 5;
   CEB2_A.delay[30] := 10;
   CEB2_A.delay[31..33] := 5;
   CEB2_A.delay[34] := 10;
   CEB2_A.delay[35..36] := 5;
   CEB2_A.delay[37] := 10;
   CEB2_A.delay[38..39] := 5;
   CEB2_A.delay[40] := 10;
   CEB2_A.delay[41] := 5;
   CEB2_A.delay[42] := 1;
   SOFT_STOP_UF1.delay[1..4] := 5;
   SOFT_STOP_UF1.delay[5] := 1;
   SOFT_STOP_UF2.delay[1..4] := 5;
   SOFT_STOP_UF2.delay[5] := 1;
END_DATA_BLOCK

DATA_BLOCK "dtAV"   // DB80
{ S7_Optimized_Access := 'FALSE' }
VERSION : 0.1
// stored: AutoNumber false, DBAccessibleFromOPCUA true, IsOnlyStoredInLoadMemory false, IsWriteProtectedInAS false
   VAR RETAIN
      DVM201 { S7_SetPoint := 'True'} : "Av";
      SOV801 { S7_SetPoint := 'True'} : "Av";
      SOV901 { S7_SetPoint := 'True'} : "Av";
      SOV902 { S7_SetPoint := 'True'} : "Av";
      SOV1301 { S7_SetPoint := 'True'} : "Av";
      SOV1302 { S7_SetPoint := 'True'} : "Av";
      SOV1303 { S7_SetPoint := 'True'} : "Av";
      DVA501 { S7_SetPoint := 'True'} : "Av";
      DVA502 { S7_SetPoint := 'True'} : "Av";
      DVA504 { S7_SetPoint := 'True'} : "Av";
      DVA505 { S7_SetPoint := 'True'} : "Av";
      DVA506 { S7_SetPoint := 'True'} : "Av";
      DVA507 { S7_SetPoint := 'True'} : "Av";
      DVA508 { S7_SetPoint := 'True'} : "Av";
      DVA509 { S7_SetPoint := 'True'} : "Av";
      DVA511 { S7_SetPoint := 'True'} : "Av";
      DVA512 { S7_SetPoint := 'True'} : "Av";
      DVA513 { S7_SetPoint := 'True'} : "Av";
      DVA514 { S7_SetPoint := 'True'} : "Av";
      DVA515 { S7_SetPoint := 'True'} : "Av";
      DVA516 { S7_SetPoint := 'True'} : "Av";
      DVA1801 { S7_SetPoint := 'True'} : "Av";
      DVA503 { S7_SetPoint := 'True'} : "Av";
      DVA510 { S7_SetPoint := 'True'} : "Av";
      MDF4 { S7_SetPoint := 'True'} : "Av";
   END_VAR
BEGIN
END_DATA_BLOCK

ORGANIZATION_BLOCK "Main"   // OB1, LAD, ProgramCycle
TITLE = "Main Program Sweep (Cycle)"
{ S7_Optimized_Access := 'TRUE' }
VERSION : 0.1
// stored: AutoNumber true, IsIECCheckEnabled false, SetENOAutomatically false
   VAR_INPUT
      Initial_Call : Bool;   // Initial call of this OB
      Remanence : Bool;   // =True, if remanent data are available
   END_VAR
BEGIN

REGION Network 1: Клапаны
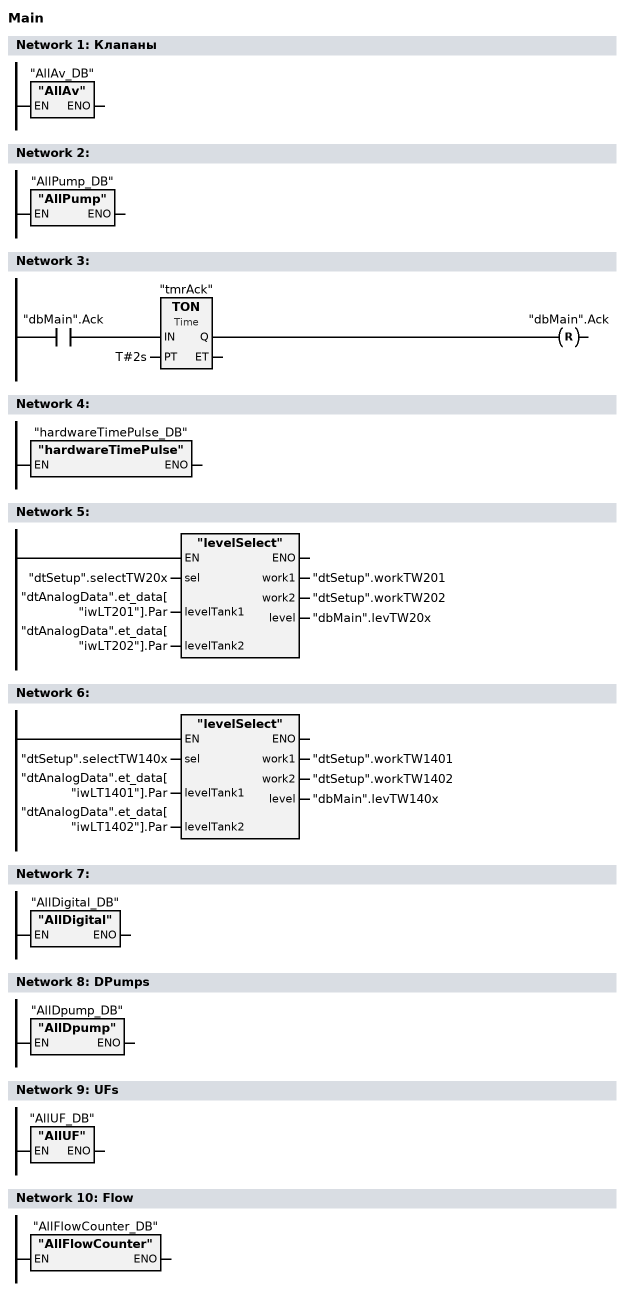
   RUNG wire#powerrail
      "AllAv_DB"()
   END_RUNG
   // the same network as SCL:
   "AllAv_DB"();   // "AllAv"
END_REGION

REGION Network 2
   RUNG wire#powerrail
      "AllPump_DB"()
   END_RUNG
   // the same network as SCL:
   "AllPump_DB"();   // "AllPump"
END_REGION

REGION Network 3
   RUNG wire#powerrail
      Contact( "dbMain".Ack )
      { S7_Templates := "time_type := Time" } "tmrAck".TON(pt := T#2s, et =>)
      R_Coil( "dbMain".Ack )
   END_RUNG
   // the same network as SCL:
   "tmrAck".TON(IN := "dbMain".Ack, PT := T#2s);
   IF "tmrAck".Q THEN "dbMain".Ack := FALSE; END_IF;
END_REGION

REGION Network 4
   RUNG wire#powerrail
      "hardwareTimePulse_DB"()
   END_RUNG
   // the same network as SCL:
   "hardwareTimePulse_DB"();   // "hardwareTimePulse"
END_REGION

REGION Network 5
   RUNG wire#powerrail
      "levelSelect"(sel := "dtSetup".selectTW20x, levelTank1 := "dtAnalogData".et_data["iwLT201"].Par, levelTank2 := "dtAnalogData".et_data["iwLT202"].Par, work1 => "dtSetup".workTW201, work2 => "dtSetup".workTW202, level => "dbMain".levTW20x)
   END_RUNG
   // the same network as SCL:
   "levelSelect"(sel := "dtSetup".selectTW20x,
                 levelTank1 := "dtAnalogData".et_data["iwLT201"].Par,
                 levelTank2 := "dtAnalogData".et_data["iwLT202"].Par,
                 work1 => "dtSetup".workTW201,
                 work2 => "dtSetup".workTW202,
                 level => "dbMain".levTW20x);
END_REGION

REGION Network 6
   RUNG wire#powerrail
      "levelSelect"(sel := "dtSetup".selectTW140x, levelTank1 := "dtAnalogData".et_data["iwLT1401"].Par, levelTank2 := "dtAnalogData".et_data["iwLT1402"].Par, work1 => "dtSetup".workTW1401, work2 => "dtSetup".workTW1402, level => "dbMain".levTW140x)
   END_RUNG
   // the same network as SCL:
   "levelSelect"(sel := "dtSetup".selectTW140x,
                 levelTank1 := "dtAnalogData".et_data["iwLT1401"].Par,
                 levelTank2 := "dtAnalogData".et_data["iwLT1402"].Par,
                 work1 => "dtSetup".workTW1401,
                 work2 => "dtSetup".workTW1402,
                 level => "dbMain".levTW140x);
END_REGION

REGION Network 7
   RUNG wire#powerrail
      "AllDigital_DB"()
   END_RUNG
   // the same network as SCL:
   "AllDigital_DB"();   // "AllDigital"
END_REGION

REGION Network 8: DPumps
   RUNG wire#powerrail
      "AllDpump_DB"()
   END_RUNG
   // the same network as SCL:
   "AllDpump_DB"();   // "AllDpump"
END_REGION

REGION Network 9: UFs
   RUNG wire#powerrail
      "AllUF_DB"()
   END_RUNG
   // the same network as SCL:
   "AllUF_DB"();   // "AllUF"
END_REGION

REGION Network 10: Flow
   RUNG wire#powerrail
      "AllFlowCounter_DB"()
   END_RUNG
   // the same network as SCL:
   "AllFlowCounter_DB"();   // "AllFlowCounter"
END_REGION
END_ORGANIZATION_BLOCK

FUNCTION_BLOCK "AllPump"   // FB2, FBD
{ S7_Optimized_Access := 'TRUE' }
VERSION : 0.1
// stored: AutoNumber true, IsIECCheckEnabled false, IsRetainMemResEnabled false, MemoryReserve 100, SetENOAutomatically false, UDAEnableTagReadback false
   VAR
      PU30x { S7_SetPoint := 'True'} : "PumpCntrl2Pu1Fc";
      cmUZ_P30x { S7_SetPoint := 'True'} : Bool;
      cmUZ_P120x : Bool;
      cmUZ_P150x : Bool;
      tmrLowPresP30x { S7_SetPoint := 'True'} : TON_TIME;
      tmrLowFreqP30x { S7_SetPoint := 'True'} : TON_TIME;
      tLowPresP30x { S7_SetPoint := 'True'} : Time;
      tLowFreqP30x : Time;
      PU120x { S7_SetPoint := 'True'} : "PumpCntrl2Pu1Fc";
      tmrLowPresP120x { S7_SetPoint := 'True'} : TON_TIME;
      tLowPresP120x { S7_SetPoint := 'True'} : Time;
      tNoPulseP120x : Time;
      PU150x { S7_SetPoint := 'True'} : "PumpCntrl2Pu1Fc";
      tmrLowPresP150x { S7_SetPoint := 'True'} : TON_TIME;
      tLowPresP150x { S7_SetPoint := 'True'} : Time;
      tNoPulseP150x : Time;
      noPulseTOF_P120x { S7_SetPoint := 'True'} : "noPulseTOF";
      noPulseTOF_P150x { S7_SetPoint := 'True'} : "noPulseTOF";
      P701 { S7_SetPoint := 'True'} : "PumpCntr";
      P702 { S7_SetPoint := 'True'} : "PumpCntr";
      P901 { S7_SetPoint := 'True'} : "PumpCntr";
      P1301 { S7_SetPoint := 'True'} : "PumpCntr";
      P2001 { S7_SetPoint := 'True'} : "PumpCntr";
      C501 { S7_SetPoint := 'True'} : "PumpCntr";
      sel2pu_P70x { S7_SetPoint := 'True'} : "sel2pu";
   END_VAR
BEGIN

REGION Network 1: P30x - выбор рабочего
   // Помилка датчиків рівня TW201, TW202
   // Аварійно низький рівень TW201, TW202
   // Помилка датчика PT301
   // Аварійно низьке значення PT301
   // Аварійно високе значення PT301
   // Помилка датчика PT401
   // Аварійно низьке значення PT401
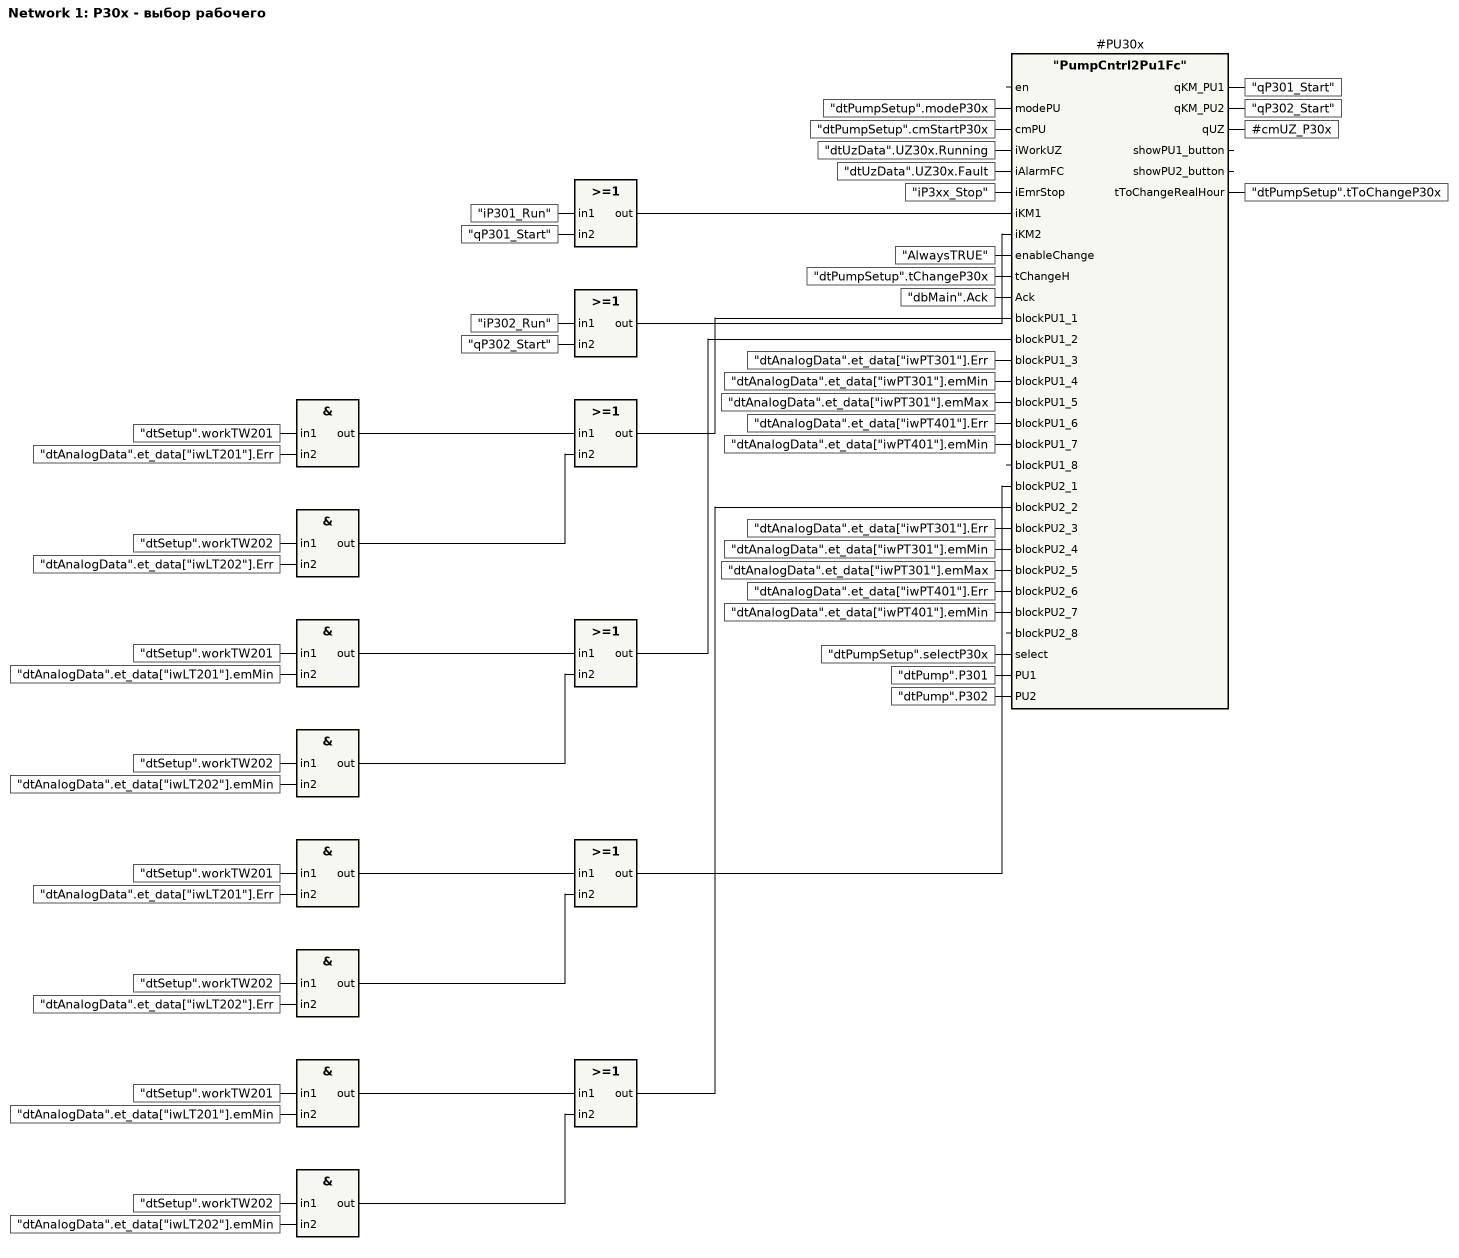
   #PU30x(modePU := "dtPumpSetup".modeP30x,   // "PumpCntrl2Pu1Fc"
          cmPU := "dtPumpSetup".cmStartP30x,
          iWorkUZ := "dtUzData".UZ30x.Running,
          iAlarmFC := "dtUzData".UZ30x.Fault,
          iEmrStop := "iP3xx_Stop",
          iKM1 := "iP301_Run" OR "qP301_Start",
          iKM2 := "iP302_Run" OR "qP302_Start",
          enableChange := "AlwaysTRUE",
          tChangeH := "dtPumpSetup".tChangeP30x,
          Ack := "dbMain".Ack,
          blockPU1_1 := ("dtSetup".workTW201 AND "dtAnalogData".et_data["iwLT201"].Err) OR ("dtSetup".workTW202 AND "dtAnalogData".et_data["iwLT202"].Err),
          blockPU1_2 := ("dtSetup".workTW201 AND "dtAnalogData".et_data["iwLT201"].emMin) OR ("dtSetup".workTW202 AND "dtAnalogData".et_data["iwLT202"].emMin),
          blockPU1_3 := "dtAnalogData".et_data["iwPT301"].Err,
          blockPU1_4 := "dtAnalogData".et_data["iwPT301"].emMin,
          blockPU1_5 := "dtAnalogData".et_data["iwPT301"].emMax,
          blockPU1_6 := "dtAnalogData".et_data["iwPT401"].Err,
          blockPU1_7 := "dtAnalogData".et_data["iwPT401"].emMin,
          blockPU2_1 := ("dtSetup".workTW201 AND "dtAnalogData".et_data["iwLT201"].Err) OR ("dtSetup".workTW202 AND "dtAnalogData".et_data["iwLT202"].Err),
          blockPU2_2 := ("dtSetup".workTW201 AND "dtAnalogData".et_data["iwLT201"].emMin) OR ("dtSetup".workTW202 AND "dtAnalogData".et_data["iwLT202"].emMin),
          blockPU2_3 := "dtAnalogData".et_data["iwPT301"].Err,
          blockPU2_4 := "dtAnalogData".et_data["iwPT301"].emMin,
          blockPU2_5 := "dtAnalogData".et_data["iwPT301"].emMax,
          blockPU2_6 := "dtAnalogData".et_data["iwPT401"].Err,
          blockPU2_7 := "dtAnalogData".et_data["iwPT401"].emMin,
          select := "dtPumpSetup".selectP30x,
          PU1 := "dtPump".P301,
          PU2 := "dtPump".P302,
          qKM_PU1 => "qP301_Start",
          qKM_PU2 => "qP302_Start",
          qUZ => #cmUZ_P30x,
          tToChangeRealHour => "dtPumpSetup".tToChangeP30x);
END_REGION

REGION Network 2: P30x - частотник
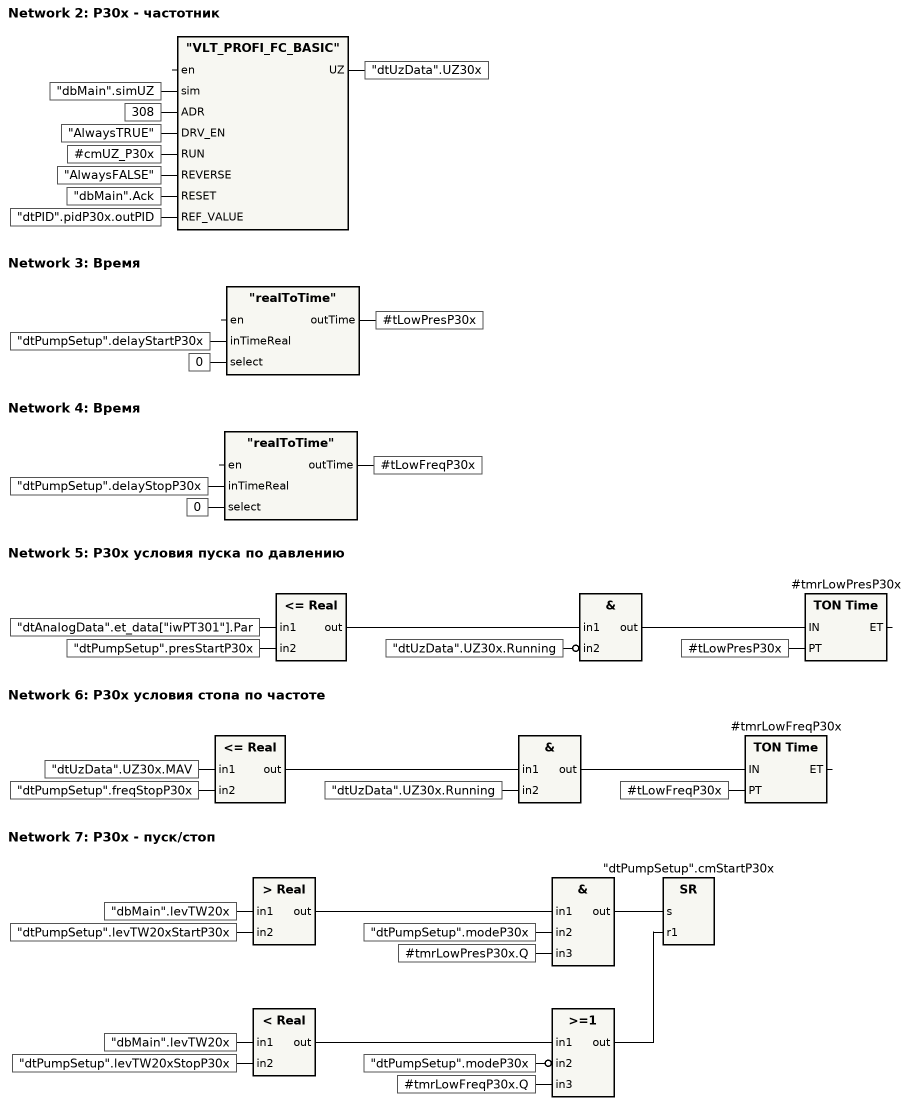
   "VLT_PROFI_FC_BASIC"(sim := "dbMain".simUZ,
                        ADR := 308,
                        DRV_EN := "AlwaysTRUE",
                        RUN := #cmUZ_P30x,
                        REVERSE := "AlwaysFALSE",
                        RESET := "dbMain".Ack,
                        REF_VALUE := "dtPID".pidP30x.outPID,
                        UZ => "dtUzData".UZ30x);
END_REGION

REGION Network 3: Время
   "realToTime"(inTimeReal := "dtPumpSetup".delayStartP30x, select := 0, outTime => #tLowPresP30x);
END_REGION

REGION Network 4: Время
   "realToTime"(inTimeReal := "dtPumpSetup".delayStopP30x, select := 0, outTime => #tLowFreqP30x);
END_REGION

REGION Network 5: P30x условия пуска по давлению
   #tmrLowPresP30x(IN := ("dtAnalogData".et_data["iwPT301"].Par <= "dtPumpSetup".presStartP30x) AND NOT "dtUzData".UZ30x.Running,   // TON
                   PT := #tLowPresP30x);
END_REGION

REGION Network 6: P30x условия стопа по частоте
   #tmrLowFreqP30x(IN := ("dtUzData".UZ30x.MAV <= "dtPumpSetup".freqStopP30x) AND "dtUzData".UZ30x.Running,   // TON
                   PT := #tLowFreqP30x);
END_REGION

REGION Network 7: P30x - пуск/стоп
   IF ("dbMain".levTW20x > "dtPumpSetup".levTW20xStartP30x) AND "dtPumpSetup".modeP30x AND #tmrLowPresP30x.Q THEN
       "dtPumpSetup".cmStartP30x := TRUE;   // SR flip-flop
   END_IF;
   IF ("dbMain".levTW20x < "dtPumpSetup".levTW20xStopP30x) OR NOT "dtPumpSetup".modeP30x OR #tmrLowFreqP30x.Q THEN
       "dtPumpSetup".cmStartP30x := FALSE;
   END_IF;
END_REGION

REGION Network 8: -------------------------------------------------P1201, 1202
END_REGION

REGION Network 9: P120x - выбор рабочего !!!!!!!!!!!!!!!!!!!!!!!!!!!!!!!!!!!!!!!!!!!!!!!!!! Убрать iP1201_run
   // Помилка датчиків рівня LT1101
   // Аварійно низький рівень TW1101
   // Помилка датчика PT1201
   // Аварійно низьке значення PT1201
   // Аварійно високе значення PT1201
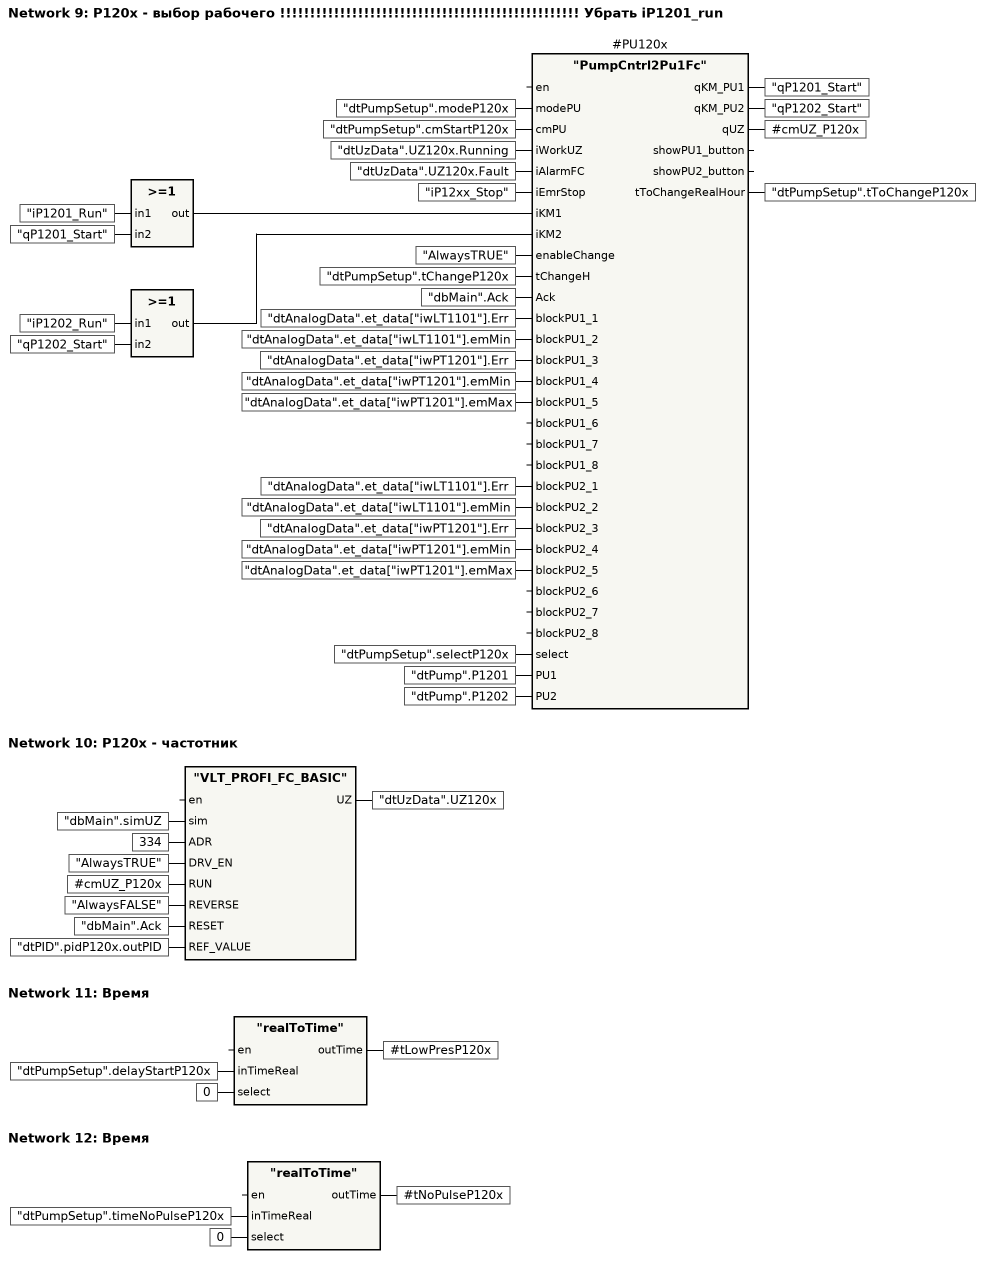
   #PU120x(modePU := "dtPumpSetup".modeP120x,   // "PumpCntrl2Pu1Fc"
           cmPU := "dtPumpSetup".cmStartP120x,
           iWorkUZ := "dtUzData".UZ120x.Running,
           iAlarmFC := "dtUzData".UZ120x.Fault,
           iEmrStop := "iP12xx_Stop",
           iKM1 := "iP1201_Run" OR "qP1201_Start",
           iKM2 := "iP1202_Run" OR "qP1202_Start",
           enableChange := "AlwaysTRUE",
           tChangeH := "dtPumpSetup".tChangeP120x,
           Ack := "dbMain".Ack,
           blockPU1_1 := "dtAnalogData".et_data["iwLT1101"].Err,
           blockPU1_2 := "dtAnalogData".et_data["iwLT1101"].emMin,
           blockPU1_3 := "dtAnalogData".et_data["iwPT1201"].Err,
           blockPU1_4 := "dtAnalogData".et_data["iwPT1201"].emMin,
           blockPU1_5 := "dtAnalogData".et_data["iwPT1201"].emMax,
           blockPU2_1 := "dtAnalogData".et_data["iwLT1101"].Err,
           blockPU2_2 := "dtAnalogData".et_data["iwLT1101"].emMin,
           blockPU2_3 := "dtAnalogData".et_data["iwPT1201"].Err,
           blockPU2_4 := "dtAnalogData".et_data["iwPT1201"].emMin,
           blockPU2_5 := "dtAnalogData".et_data["iwPT1201"].emMax,
           select := "dtPumpSetup".selectP120x,
           PU1 := "dtPump".P1201,
           PU2 := "dtPump".P1202,
           qKM_PU1 => "qP1201_Start",
           qKM_PU2 => "qP1202_Start",
           qUZ => #cmUZ_P120x,
           tToChangeRealHour => "dtPumpSetup".tToChangeP120x);
END_REGION

REGION Network 10: P120x - частотник
   "VLT_PROFI_FC_BASIC"(sim := "dbMain".simUZ,
                        ADR := 334,
                        DRV_EN := "AlwaysTRUE",
                        RUN := #cmUZ_P120x,
                        REVERSE := "AlwaysFALSE",
                        RESET := "dbMain".Ack,
                        REF_VALUE := "dtPID".pidP120x.outPID,
                        UZ => "dtUzData".UZ120x);
END_REGION

REGION Network 11: Время
   "realToTime"(inTimeReal := "dtPumpSetup".delayStartP120x, select := 0, outTime => #tLowPresP120x);
END_REGION

REGION Network 12: Время
   "realToTime"(inTimeReal := "dtPumpSetup".timeNoPulseP120x, select := 0, outTime => #tNoPulseP120x);
END_REGION

REGION Network 13: P120x условия пуска по давлению
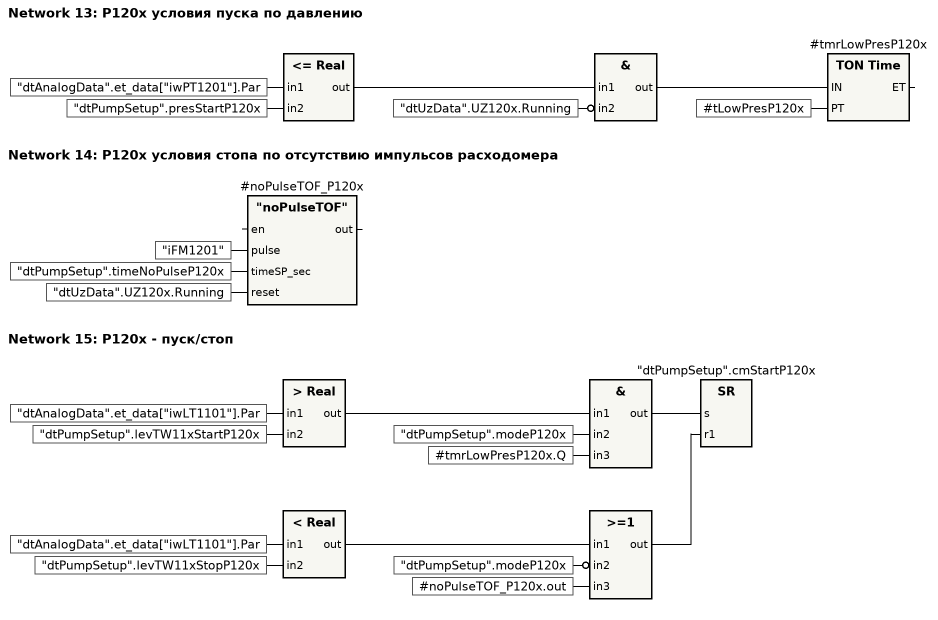
   #tmrLowPresP120x(IN := ("dtAnalogData".et_data["iwPT1201"].Par <= "dtPumpSetup".presStartP120x) AND NOT "dtUzData".UZ120x.Running,   // TON
                    PT := #tLowPresP120x);
END_REGION

REGION Network 14: P120x условия стопа по отсутствию импульсов расходомера
   #noPulseTOF_P120x(pulse := "iFM1201",   // "noPulseTOF"
                     timeSP_sec := "dtPumpSetup".timeNoPulseP120x,
                     reset := "dtUzData".UZ120x.Running);
END_REGION

REGION Network 15: P120x - пуск/стоп
   IF ("dtAnalogData".et_data["iwLT1101"].Par > "dtPumpSetup".levTW11xStartP120x) AND "dtPumpSetup".modeP120x AND #tmrLowPresP120x.Q THEN
       "dtPumpSetup".cmStartP120x := TRUE;   // SR flip-flop
   END_IF;
   IF ("dtAnalogData".et_data["iwLT1101"].Par < "dtPumpSetup".levTW11xStopP120x) OR NOT "dtPumpSetup".modeP120x OR #noPulseTOF_P120x.out THEN
       "dtPumpSetup".cmStartP120x := FALSE;
   END_IF;
END_REGION

REGION Network 16: -------------------------------------------------P1501, 1502
END_REGION

REGION Network 17: P150x - выбор рабочего !!!!!!!!!!!!!!!!!!!!!!!!!!!!!!!!!!!!!!!!!!!!!!!!!! Убрать iP1501_run
   // Помилка датчиків рівня TW1401, TW1402
   // Аварійно низький рівень TW1401, TW1402
   // Помилка датчика PT1501
   // Аварійно низьке значення PT1501
   // Аварійно високе значення PT1501
   // Помилка датчика PT1701
   // Аварійно низьке значення PT1701
   // Аварійно високе значення PT1701
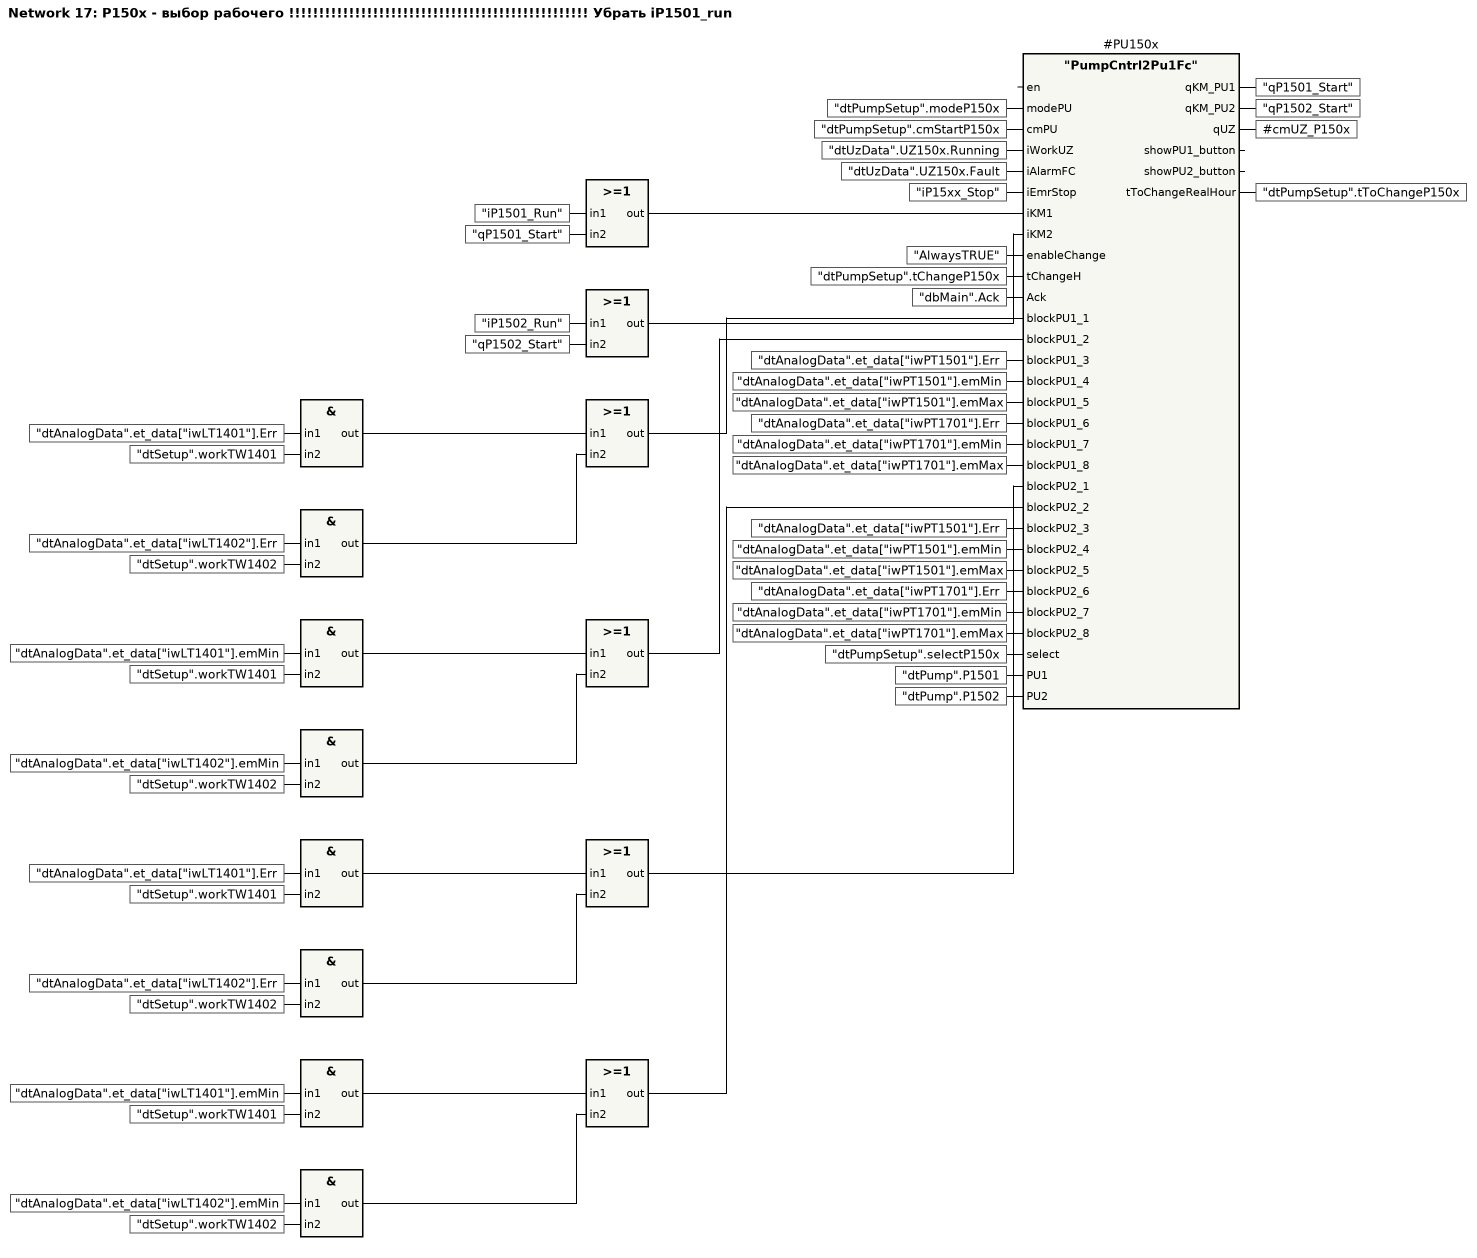
   #PU150x(modePU := "dtPumpSetup".modeP150x,   // "PumpCntrl2Pu1Fc"
           cmPU := "dtPumpSetup".cmStartP150x,
           iWorkUZ := "dtUzData".UZ150x.Running,
           iAlarmFC := "dtUzData".UZ150x.Fault,
           iEmrStop := "iP15xx_Stop",
           iKM1 := "iP1501_Run" OR "qP1501_Start",
           iKM2 := "iP1502_Run" OR "qP1502_Start",
           enableChange := "AlwaysTRUE",
           tChangeH := "dtPumpSetup".tChangeP150x,
           Ack := "dbMain".Ack,
           blockPU1_1 := ("dtAnalogData".et_data["iwLT1401"].Err AND "dtSetup".workTW1401) OR ("dtAnalogData".et_data["iwLT1402"].Err AND "dtSetup".workTW1402),
           blockPU1_2 := ("dtAnalogData".et_data["iwLT1401"].emMin AND "dtSetup".workTW1401) OR ("dtAnalogData".et_data["iwLT1402"].emMin AND "dtSetup".workTW1402),
           blockPU1_3 := "dtAnalogData".et_data["iwPT1501"].Err,
           blockPU1_4 := "dtAnalogData".et_data["iwPT1501"].emMin,
           blockPU1_5 := "dtAnalogData".et_data["iwPT1501"].emMax,
           blockPU1_6 := "dtAnalogData".et_data["iwPT1701"].Err,
           blockPU1_7 := "dtAnalogData".et_data["iwPT1701"].emMin,
           blockPU1_8 := "dtAnalogData".et_data["iwPT1701"].emMax,
           blockPU2_1 := ("dtAnalogData".et_data["iwLT1401"].Err AND "dtSetup".workTW1401) OR ("dtAnalogData".et_data["iwLT1402"].Err AND "dtSetup".workTW1402),
           blockPU2_2 := ("dtAnalogData".et_data["iwLT1401"].emMin AND "dtSetup".workTW1401) OR ("dtAnalogData".et_data["iwLT1402"].emMin AND "dtSetup".workTW1402),
           blockPU2_3 := "dtAnalogData".et_data["iwPT1501"].Err,
           blockPU2_4 := "dtAnalogData".et_data["iwPT1501"].emMin,
           blockPU2_5 := "dtAnalogData".et_data["iwPT1501"].emMax,
           blockPU2_6 := "dtAnalogData".et_data["iwPT1701"].Err,
           blockPU2_7 := "dtAnalogData".et_data["iwPT1701"].emMin,
           blockPU2_8 := "dtAnalogData".et_data["iwPT1701"].emMax,
           select := "dtPumpSetup".selectP150x,
           PU1 := "dtPump".P1501,
           PU2 := "dtPump".P1502,
           qKM_PU1 => "qP1501_Start",
           qKM_PU2 => "qP1502_Start",
           qUZ => #cmUZ_P150x,
           tToChangeRealHour => "dtPumpSetup".tToChangeP150x);
END_REGION

REGION Network 18: P150x - частотник
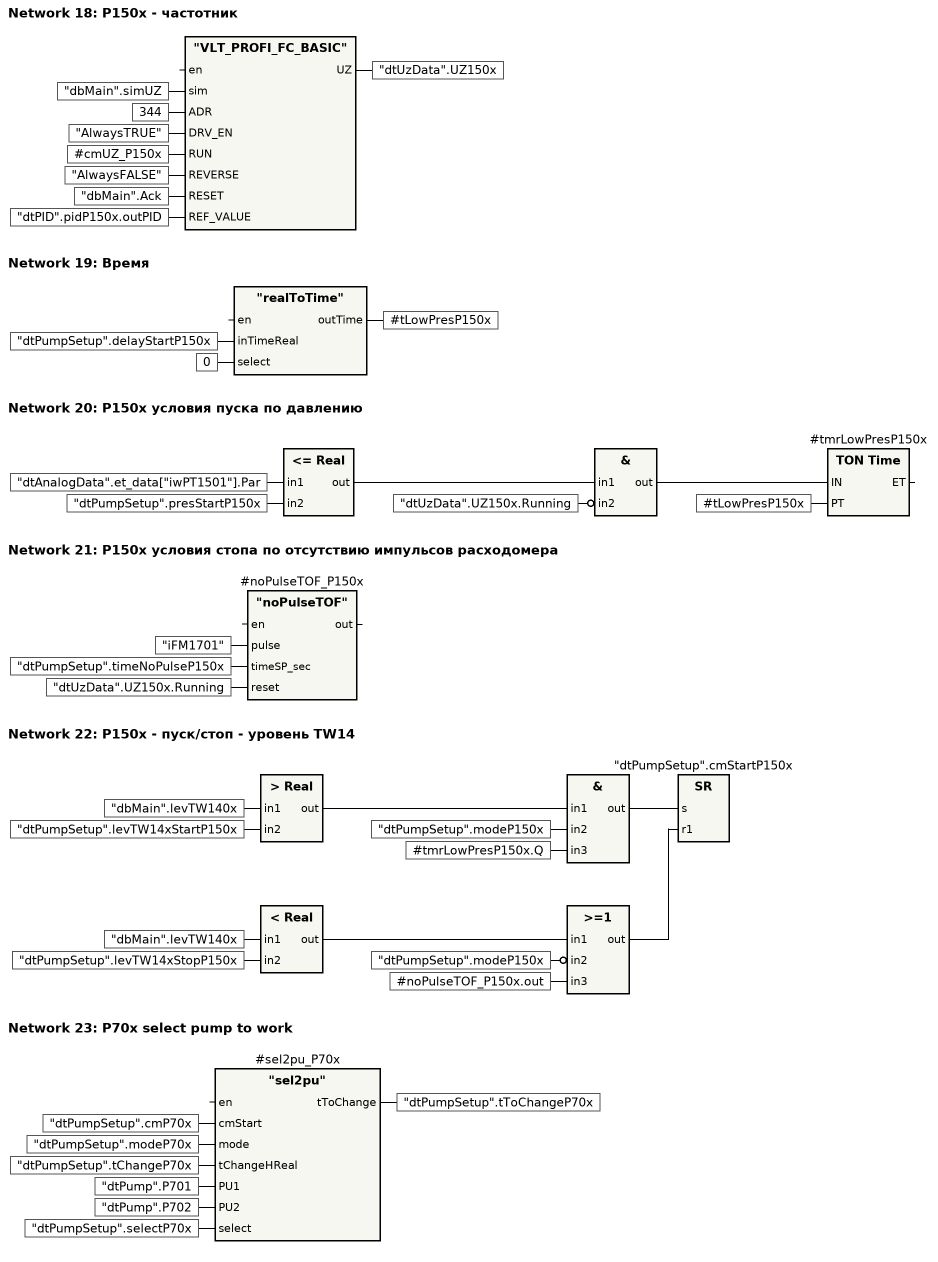
   "VLT_PROFI_FC_BASIC"(sim := "dbMain".simUZ,
                        ADR := 344,
                        DRV_EN := "AlwaysTRUE",
                        RUN := #cmUZ_P150x,
                        REVERSE := "AlwaysFALSE",
                        RESET := "dbMain".Ack,
                        REF_VALUE := "dtPID".pidP150x.outPID,
                        UZ => "dtUzData".UZ150x);
END_REGION

REGION Network 19: Время
   "realToTime"(inTimeReal := "dtPumpSetup".delayStartP150x, select := 0, outTime => #tLowPresP150x);
END_REGION

REGION Network 20: P150x условия пуска по давлению
   #tmrLowPresP150x(IN := ("dtAnalogData".et_data["iwPT1501"].Par <= "dtPumpSetup".presStartP150x) AND NOT "dtUzData".UZ150x.Running,   // TON
                    PT := #tLowPresP150x);
END_REGION

REGION Network 21: P150x условия стопа по отсутствию импульсов расходомера
   #noPulseTOF_P150x(pulse := "iFM1701",   // "noPulseTOF"
                     timeSP_sec := "dtPumpSetup".timeNoPulseP150x,
                     reset := "dtUzData".UZ150x.Running);
END_REGION

REGION Network 22: P150x - пуск/стоп - уровень TW14
   IF ("dbMain".levTW140x > "dtPumpSetup".levTW14xStartP150x) AND "dtPumpSetup".modeP150x AND #tmrLowPresP150x.Q THEN
       "dtPumpSetup".cmStartP150x := TRUE;   // SR flip-flop
   END_IF;
   IF ("dbMain".levTW140x < "dtPumpSetup".levTW14xStopP150x) OR NOT "dtPumpSetup".modeP150x OR #noPulseTOF_P150x.out THEN
       "dtPumpSetup".cmStartP150x := FALSE;
   END_IF;
END_REGION

REGION Network 23: P70x select pump to work
   #sel2pu_P70x(cmStart := "dtPumpSetup".cmP70x,   // "sel2pu"
                mode := "dtPumpSetup".modeP70x,
                tChangeHReal := "dtPumpSetup".tChangeP70x,
                PU1 := "dtPump".P701,
                PU2 := "dtPump".P702,
                select := "dtPumpSetup".selectP70x,
                tToChange => "dtPumpSetup".tToChangeP70x);
END_REGION

REGION Network 24: P701
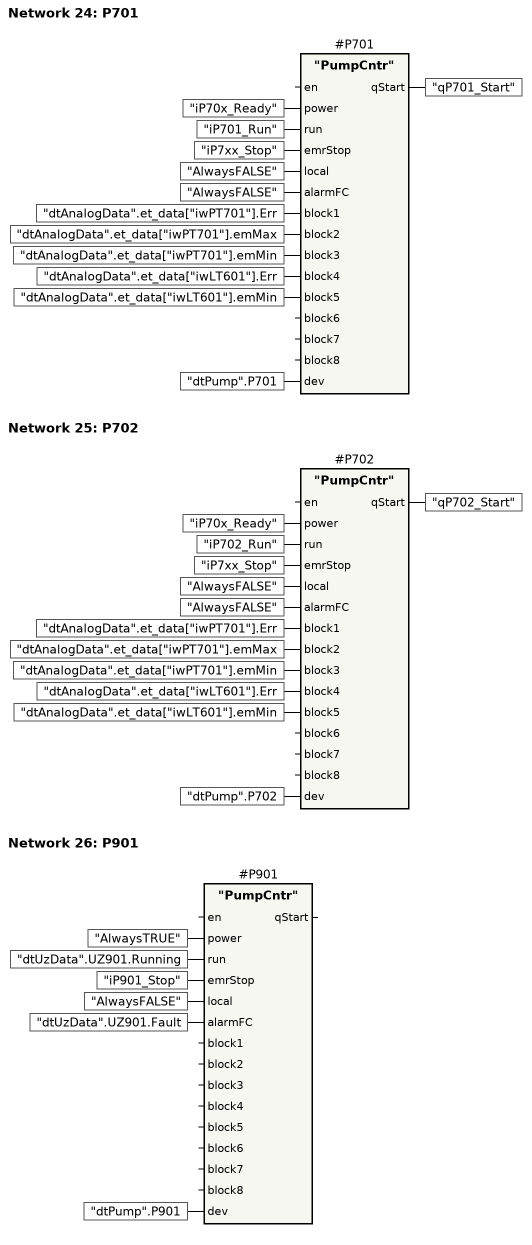
   #P701(power := "iP70x_Ready",   // "PumpCntr"
         run := "iP701_Run",
         emrStop := "iP7xx_Stop",
         local := "AlwaysFALSE",
         alarmFC := "AlwaysFALSE",
         block1 := "dtAnalogData".et_data["iwPT701"].Err,
         block2 := "dtAnalogData".et_data["iwPT701"].emMax,
         block3 := "dtAnalogData".et_data["iwPT701"].emMin,
         block4 := "dtAnalogData".et_data["iwLT601"].Err,
         block5 := "dtAnalogData".et_data["iwLT601"].emMin,
         dev := "dtPump".P701,
         qStart => "qP701_Start");
END_REGION

REGION Network 25: P702
   #P702(power := "iP70x_Ready",   // "PumpCntr"
         run := "iP702_Run",
         emrStop := "iP7xx_Stop",
         local := "AlwaysFALSE",
         alarmFC := "AlwaysFALSE",
         block1 := "dtAnalogData".et_data["iwPT701"].Err,
         block2 := "dtAnalogData".et_data["iwPT701"].emMax,
         block3 := "dtAnalogData".et_data["iwPT701"].emMin,
         block4 := "dtAnalogData".et_data["iwLT601"].Err,
         block5 := "dtAnalogData".et_data["iwLT601"].emMin,
         dev := "dtPump".P702,
         qStart => "qP702_Start");
END_REGION

REGION Network 26: P901
   #P901(power := "AlwaysTRUE",   // "PumpCntr"
         run := "dtUzData".UZ901.Running,
         emrStop := "iP901_Stop",
         local := "AlwaysFALSE",
         alarmFC := "dtUzData".UZ901.Fault,
         dev := "dtPump".P901);
END_REGION

REGION Network 27: P901 - частотник
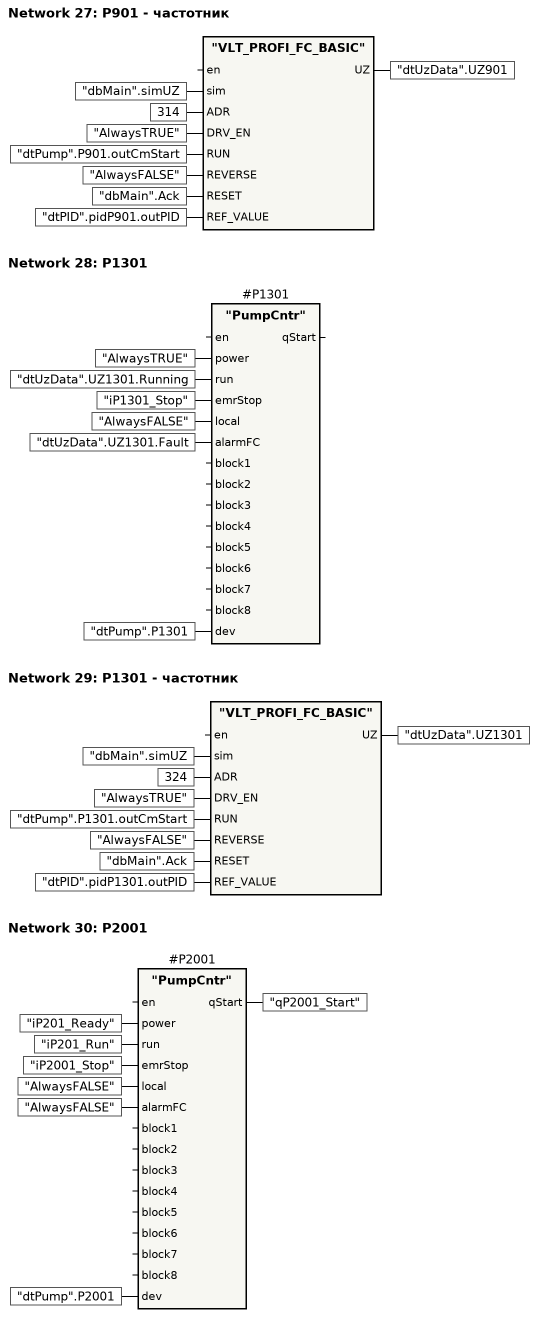
   "VLT_PROFI_FC_BASIC"(sim := "dbMain".simUZ,
                        ADR := 314,
                        DRV_EN := "AlwaysTRUE",
                        RUN := "dtPump".P901.outCmStart,
                        REVERSE := "AlwaysFALSE",
                        RESET := "dbMain".Ack,
                        REF_VALUE := "dtPID".pidP901.outPID,
                        UZ => "dtUzData".UZ901);
END_REGION

REGION Network 28: P1301
   #P1301(power := "AlwaysTRUE",   // "PumpCntr"
          run := "dtUzData".UZ1301.Running,
          emrStop := "iP1301_Stop",
          local := "AlwaysFALSE",
          alarmFC := "dtUzData".UZ1301.Fault,
          dev := "dtPump".P1301);
END_REGION

REGION Network 29: P1301 - частотник
   "VLT_PROFI_FC_BASIC"(sim := "dbMain".simUZ,
                        ADR := 324,
                        DRV_EN := "AlwaysTRUE",
                        RUN := "dtPump".P1301.outCmStart,
                        REVERSE := "AlwaysFALSE",
                        RESET := "dbMain".Ack,
                        REF_VALUE := "dtPID".pidP1301.outPID,
                        UZ => "dtUzData".UZ1301);
END_REGION

REGION Network 30: P2001
   #P2001(power := "iP201_Ready",   // "PumpCntr"
          run := "iP201_Run",
          emrStop := "iP2001_Stop",
          local := "AlwaysFALSE",
          alarmFC := "AlwaysFALSE",
          dev := "dtPump".P2001,
          qStart => "qP2001_Start");
END_REGION
END_FUNCTION_BLOCK

FUNCTION_BLOCK "PumpCntrl2Pu1Fc"   // FB61, FBD
{ S7_Optimized_Access := 'TRUE' }
VERSION : 0.1
// 0 0 -стоп, 1- работа
// 1 2 - Запуск
// 2 4 - Остановка
// 3 8 - Сервисный режим
// 4 16 - Ошибка пуска
// 5 32 - Ошибка останова
// 6 64 - Ошибка питания
// 7 128 - Ошибка Частотника
// 8 256 - Блокировка внешняя (сборная)
// 9 - 512 - Нажат аварийный стоп
// 10 -U24 - Сборная авария
// 11 - 2048 - Местный режим
// 12 -  4096 - Ошибка вклчюния контактора
// 13 - 8192 - шбика отключения контактора
// 14 -  16384 - 1 показывать кнопки ручного управления
// 15 - 32768 - режим 1-ручной, 0-авто (только для индикатора на скаде)
// stored: AutoNumber false, IsIECCheckEnabled false, IsRetainMemResEnabled false, MemoryReserve 100, SetENOAutomatically false, UDAEnableTagReadback false
   VAR_INPUT
      modePU : Bool;
      cmPU : Bool;
      iWorkUZ : Bool;
      iAlarmFC : Bool;
      iEmrStop : Bool;
      iKM1 : Bool;
      iKM2 : Bool;
      enableChange : Bool;
      tChangeH : Real;
      Ack : Bool;
      blockPU1_1 : Bool;
      blockPU1_2 : Bool;
      blockPU1_3 : Bool;
      blockPU1_4 : Bool;
      blockPU1_5 : Bool;
      blockPU1_6 : Bool;
      blockPU1_7 : Bool;
      blockPU1_8 : Bool;
      blockPU2_1 : Bool;
      blockPU2_2 : Bool;
      blockPU2_3 : Bool;
      blockPU2_4 : Bool;
      blockPU2_5 : Bool;
      blockPU2_6 : Bool;
      blockPU2_7 : Bool;
      blockPU2_8 : Bool;
   END_VAR
   VAR_OUTPUT
      qKM_PU1 : Bool;
      qKM_PU2 : Bool;
      qUZ : Bool;
      showPU1_button : Bool;
      showPU2_button : Bool;
      tToChangeRealHour : Real;
   END_VAR
   VAR_IN_OUT
      select : Bool;
      PU1 : "Pump";
      PU2 : "Pump";
   END_VAR
   VAR
      cmPU1 : Bool;   // Врутренняя команда первого насоса
      cmPU2 : Bool;   // Врутренняя команда второго насоса
      selectInternal : Bool;
      TOFcmPU1 { S7_SetPoint := 'True'} : TOF_TIME;
      TOFcmPU2 { S7_SetPoint := 'True'} : TOF_TIME;
   END_VAR
   VAR RETAIN
      tWork1 : DInt;
      tWork2 : DInt;
   END_VAR
   VAR
      tChange : DInt;
      needChange : Bool;
      tmpDInt : DInt;
      errAlarmFC_PU1 : Bool;
      errAlarmFC_PU2 : Bool;
      errBlock_PU1 : Bool;
      errBlock_PU2 : Bool;
      tmrErrOnUZ : TON_TIME;
      errON_UZ_PU1 : Bool;
      errON_UZ_PU2 : Bool;
      tmrErrOffUZ : TON_TIME;
      errOff_UZ_PU1 : Bool;
      errOff_UZ_PU2 : Bool;
      tmrErrOnKM_PU1 : TON_TIME;
      errOn_KM_PU1 : Bool;
      errOn_KM_PU2 : Bool;
      errOff_KM_PU1 : Bool;
      errOff_KM_PU2 : Bool;
      tmrErrOnKM_PU2 { S7_SetPoint := 'True'} : TON_TIME;
      tmrErrOffKM_PU1 { S7_SetPoint := 'True'} : TON_TIME;
      tmrErrOffKM_PU2 { S7_SetPoint := 'True'} : TON_TIME;
      errServicePU1 : Bool;
      errServicePU2 : Bool;
      tStartPU_FC : Time;
      tStopPU_FC : Time;
      tToChangeDint : DInt;
      errEmrStopPU1 : Bool;
      errEmrStopPU2 : Bool;
   END_VAR
BEGIN

REGION Network 1: Режим
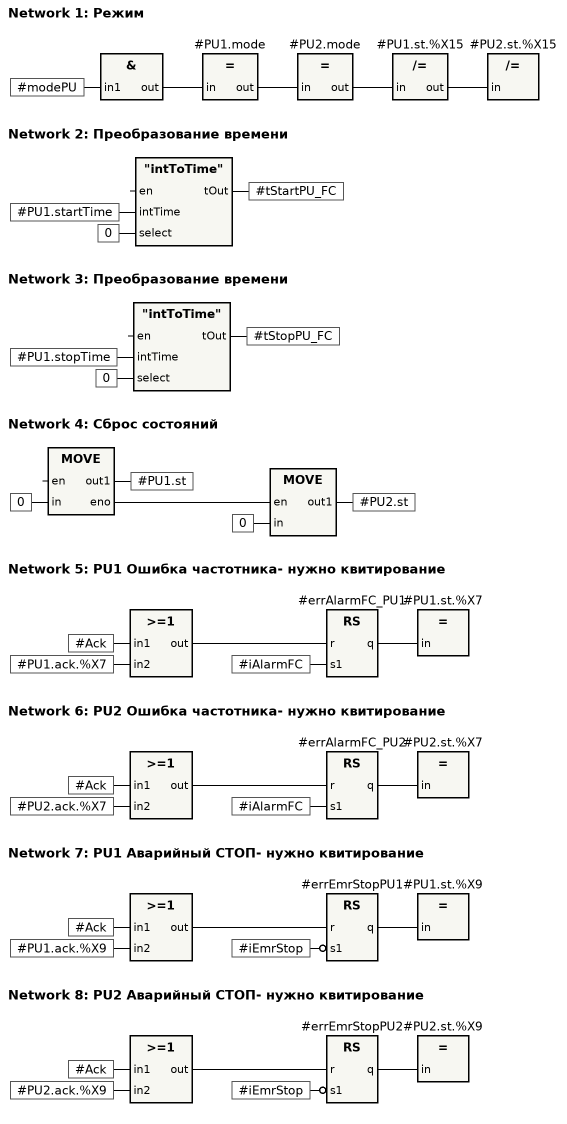
   #PU1.mode := #modePU;
   #PU2.mode := #modePU;
   #PU1.st.%X15 := NOT #modePU;
   #PU2.st.%X15 := NOT #modePU;
END_REGION

REGION Network 2: Преобразование времени
   // ВРемя из настроек первого насоса
   "intToTime"(intTime := #PU1.startTime, select := 0, tOut => #tStartPU_FC);
END_REGION

REGION Network 3: Преобразование времени
   // ВРемя из настроек первого насоса
   "intToTime"(intTime := #PU1.stopTime, select := 0, tOut => #tStopPU_FC);
END_REGION

REGION Network 4: Сброс состояний
   #PU1.st := 0;
   #PU2.st := 0;
END_REGION

REGION Network 5: PU1 Ошибка частотника- нужно квитирование
   IF #Ack OR #PU1.ack.%X7 THEN
       #errAlarmFC_PU1 := FALSE;   // RS flip-flop
   END_IF;
   IF #iAlarmFC THEN #errAlarmFC_PU1 := TRUE; END_IF;
   #PU1.st.%X7 := #errAlarmFC_PU1;
END_REGION

REGION Network 6: PU2 Ошибка частотника- нужно квитирование
   IF #Ack OR #PU2.ack.%X7 THEN
       #errAlarmFC_PU2 := FALSE;   // RS flip-flop
   END_IF;
   IF #iAlarmFC THEN #errAlarmFC_PU2 := TRUE; END_IF;
   #PU2.st.%X7 := #errAlarmFC_PU2;
END_REGION

REGION Network 7: PU1 Аварийный СТОП- нужно квитирование
   IF #Ack OR #PU1.ack.%X9 THEN
       #errEmrStopPU1 := FALSE;   // RS flip-flop
   END_IF;
   IF NOT #iEmrStop THEN #errEmrStopPU1 := TRUE; END_IF;
   #PU1.st.%X9 := #errEmrStopPU1;
END_REGION

REGION Network 8: PU2 Аварийный СТОП- нужно квитирование
   IF #Ack OR #PU2.ack.%X9 THEN
       #errEmrStopPU2 := FALSE;   // RS flip-flop
   END_IF;
   IF NOT #iEmrStop THEN #errEmrStopPU2 := TRUE; END_IF;
   #PU2.st.%X9 := #errEmrStopPU2;
END_REGION

REGION Network 9: PU1 Внешняя блокировка - нужно квитирование
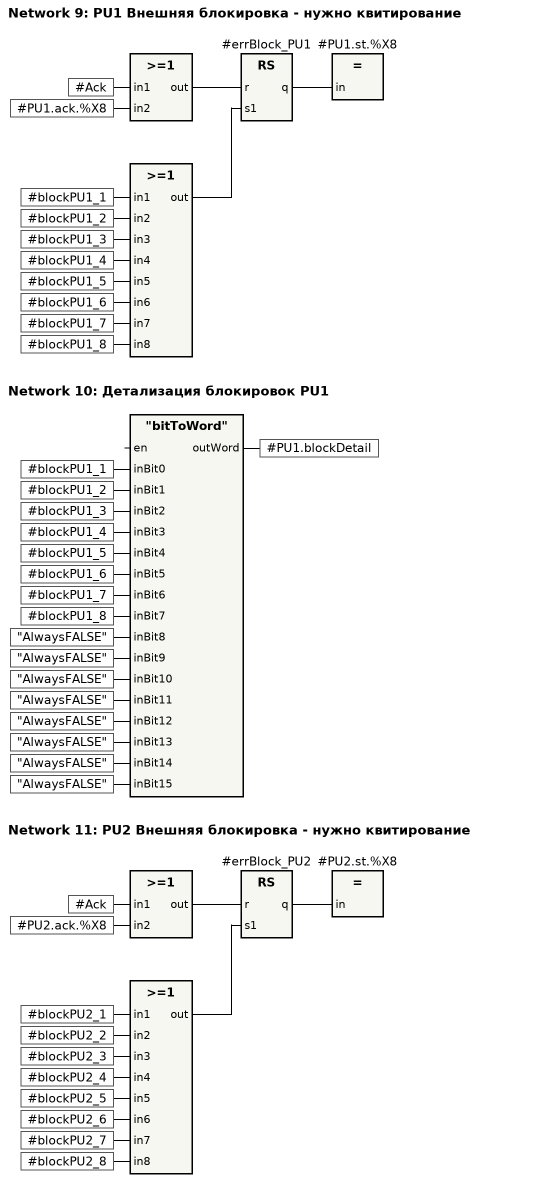
   IF #Ack OR #PU1.ack.%X8 THEN
       #errBlock_PU1 := FALSE;   // RS flip-flop
   END_IF;
   IF #blockPU1_1 OR #blockPU1_2 OR #blockPU1_3 OR #blockPU1_4 OR #blockPU1_5 OR #blockPU1_6 OR #blockPU1_7 OR #blockPU1_8 THEN
       #errBlock_PU1 := TRUE;
   END_IF;
   #PU1.st.%X8 := #errBlock_PU1;
END_REGION

REGION Network 10: Детализация блокировок PU1
   "bitToWord"(inBit0 := #blockPU1_1,
               inBit1 := #blockPU1_2,
               inBit2 := #blockPU1_3,
               inBit3 := #blockPU1_4,
               inBit4 := #blockPU1_5,
               inBit5 := #blockPU1_6,
               inBit6 := #blockPU1_7,
               inBit7 := #blockPU1_8,
               inBit8 := "AlwaysFALSE",
               inBit9 := "AlwaysFALSE",
               inBit10 := "AlwaysFALSE",
               inBit11 := "AlwaysFALSE",
               inBit12 := "AlwaysFALSE",
               inBit13 := "AlwaysFALSE",
               inBit14 := "AlwaysFALSE",
               inBit15 := "AlwaysFALSE",
               outWord => #PU1.blockDetail);
END_REGION

REGION Network 11: PU2 Внешняя блокировка - нужно квитирование
   IF #Ack OR #PU2.ack.%X8 THEN
       #errBlock_PU2 := FALSE;   // RS flip-flop
   END_IF;
   IF #blockPU2_1 OR #blockPU2_2 OR #blockPU2_3 OR #blockPU2_4 OR #blockPU2_5 OR #blockPU2_6 OR #blockPU2_7 OR #blockPU2_8 THEN
       #errBlock_PU2 := TRUE;
   END_IF;
   #PU2.st.%X8 := #errBlock_PU2;
END_REGION

REGION Network 12: Детализация блокировок PU2
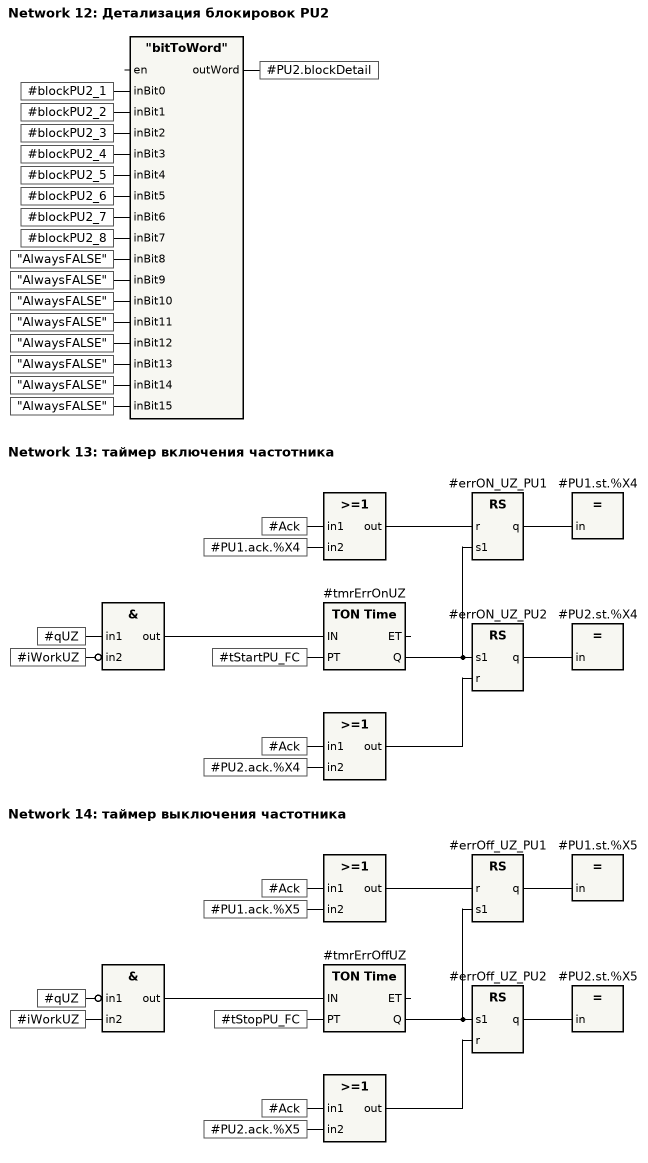
   "bitToWord"(inBit0 := #blockPU2_1,
               inBit1 := #blockPU2_2,
               inBit2 := #blockPU2_3,
               inBit3 := #blockPU2_4,
               inBit4 := #blockPU2_5,
               inBit5 := #blockPU2_6,
               inBit6 := #blockPU2_7,
               inBit7 := #blockPU2_8,
               inBit8 := "AlwaysFALSE",
               inBit9 := "AlwaysFALSE",
               inBit10 := "AlwaysFALSE",
               inBit11 := "AlwaysFALSE",
               inBit12 := "AlwaysFALSE",
               inBit13 := "AlwaysFALSE",
               inBit14 := "AlwaysFALSE",
               inBit15 := "AlwaysFALSE",
               outWord => #PU2.blockDetail);
END_REGION

REGION Network 13: таймер включения частотника
   #tmrErrOnUZ(IN := #qUZ AND NOT #iWorkUZ, PT := #tStartPU_FC);   // TON
   IF #Ack OR #PU1.ack.%X4 THEN
       #errON_UZ_PU1 := FALSE;   // RS flip-flop
   END_IF;
   IF #tmrErrOnUZ.Q THEN #errON_UZ_PU1 := TRUE; END_IF;
   #PU1.st.%X4 := #errON_UZ_PU1;
   IF #Ack OR #PU2.ack.%X4 THEN
       #errON_UZ_PU2 := FALSE;   // RS flip-flop
   END_IF;
   IF #tmrErrOnUZ.Q THEN #errON_UZ_PU2 := TRUE; END_IF;
   #PU2.st.%X4 := #errON_UZ_PU2;
END_REGION

